// TwinCAT 3 PLC project PressTests
// Title: PressTests
// Company: fraktal-automation
// Author: fraktal-automation
// ProjectVersion: 0.1.0.1
// Description: Press example TcUnit gate - excluded from deployed runtime (Core 5.7).
// ProgramVersion: 3.1.4026.24
// libraries:
//   Tc2_Standard, * (Beckhoff Automation GmbH)
//   Tc2_System, * (Beckhoff Automation GmbH)
//   Tc2_Utilities, * (Beckhoff Automation GmbH)
//   Tc3_Module, * (Beckhoff Automation GmbH)
//   Fraktal_Core, 0.25.0.0 (fraktal-automation)
//   Tc2_MC2, * (Beckhoff Automation GmbH)
//   Fraktal_Modules, 0.11.0.3 (fraktal-automation)
//   TcUnit, * (www.tcunit.org)
// project tree:
//   PressTests/ PlcTask.TcTTO, PRG_PressTestRunner.TcPOU, FB_PressDemoUnit_Tests.TcPOU, FB_FaultRecovery_Tests.TcPOU
//   Fraktal_Press_Demo/01_PneumaticPress/DUTs/ ST_PneumaticPressParCfg.TcDUT, ST_PneumaticPressStationCfg.TcDUT, ST_PneumaticPressParCmd.TcDUT (not stored), ST_PneumaticPressOutCmd.TcDUT, ST_PneumaticPressOutImm.TcDUT, E_RenditionLanguage.TcDUT, ST_PressDemoReleaseConditions.TcDUT
//   Fraktal_Press_Demo/01_PneumaticPress/ PL_PressReasons.TcGVL, FB_PressDemoUnit.TcPOU
//   Fraktal_Press_Demo/01_PneumaticPress/Recipes/ FB_PressRecipeCatalog.TcPOU
//   Fraktal_Press_Demo/01_PneumaticPress/Release/ FB_PressDemoRelease.TcPOU, FB_LD_PressDemoRelease.TcPOU, FB_PressDemoReleaseState.TcPOU
//   Fraktal_Press_Demo/01_PneumaticPress/Sequences/ FB_PressDemoHome.TcPOU, FB_PressDemoAuto.TcPOU, FB_SFC_PressDemoAuto.TcPOU, FB_LD_PressDemoAuto.TcPOU, FB_PressDemoChangeover.TcPOU, FB_PressDemoLoadPosition.TcPOU
//   Fraktal_Press_Demo/01_PneumaticPress/Io/ GVL_PressFieldbus.TcGVL, FB_PressIoCatalog.TcPOU
// real-time tasks:
//   TASK PlcTask: cycle T#10ms, priority 20, ADS port 350

CONFIGURATION PressTests
    RESOURCE PLC ON TwinCAT3
        TASK PlcTask(INTERVAL := T#10ms, PRIORITY := 20);
        PROGRAM PRG_PressTestRunner WITH PlcTask : PRG_PressTestRunner;
    END_RESOURCE
END_CONFIGURATION

// ---- Fraktal_Press_Demo/01_PneumaticPress/DUTs/ST_PneumaticPressParCfg.TcDUT
// Core §3.8 ParCfg (SchemaVersion first; adding a member = schema change).
// v2 adds the §8.11 performance references: per-model ideal cycle (OEE
// Performance denominator, §8.5.1) and the WORK-time degradation baseline
// (§8.11.4(d); 0 = watch off).
//
// v3 REMOVES RequireTwoHandStart. It was recipe data in name only - every one of
// the four catalog records set it TRUE - and §3.8a's test is whether the value
// changes with the model. It does not: it answers whether this CELL's risk
// assessment demands a two-hand start, which is deployment data and now lives in
// ST_PneumaticPressStationCfg. A recipe that could switch it off would let a
// changeover quietly remove a required operator protection.
//
// TransferSettleTime deliberately STAYED. Its catalog values genuinely differ per
// model (80/100/120/150 ms): a heavier steel blank settles on the slide more
// slowly than a plastic one, so it is a fact about the part, not the mechanism.
TYPE ST_PneumaticPressParCfg :
STRUCT
    SchemaVersion       : UINT := 3;
    PressSettleTime     : TIME := T#500MS;
    TransferSettleTime  : TIME := T#100MS;
    IdealCycleMs        : UDINT := 0;    // §8.5.1 — 0 = Performance not computed
    BaselineWorkMs      : UDINT := 0;    // §8.11.4(d) — 0 = degradation watch off
END_STRUCT
END_TYPE

// ---- Fraktal_Press_Demo/01_PneumaticPress/DUTs/ST_PneumaticPressStationCfg.TcDUT
// Core §3.8a/§3.8b — what this PRESS is, as opposed to what the current product
// needs. Both members were assessed against one question: does the value change
// when the MODEL changes?
//
//   RequireTwoHandStart came OUT of ST_PneumaticPressParCfg. It was recipe data
//   in name only - all four catalog records set it TRUE - and it answers a
//   question about the CELL: does this installation's risk assessment demand a
//   two-hand start? A model recipe able to switch it off would let a changeover
//   quietly remove a required operator protection, which is not a decision a
//   product record should be able to take. (The certified two-hand evaluation
//   stays in TwinSAFE regardless, §9.8; this flag selects whether the AUTO cycle
//   WAITS for it, and can never weaken the safety function itself.)
//
//   StallGuardMs is the step guard for a step that declares no ExpectedTime
//   (§6.9). How long a pneumatic motion may take before it counts as stalled is
//   a fact about this machine's cylinders and air supply, not about the part.
//
// SchemaVersion is FIRST and mandatory (§3.8b). Version 0 means never written, so
// a first boot initializes silently; any other unrecognized version means a real
// image was rejected, and FB_ModuleBase.M_RestoreStationCfg reports it for the
// root to annunciate with this Unit's canonical path.
TYPE ST_PneumaticPressStationCfg :
STRUCT
    SchemaVersion       : UINT;    // 0 = never written; 1 = this layout
    RequireTwoHandStart : BOOL;    // cell risk-assessment policy, not recipe data
    StallGuardMs        : UDINT;   // §6.9 step guard when a step declares none
END_STRUCT
END_TYPE

// ---- Fraktal_Press_Demo/01_PneumaticPress/DUTs/ST_PneumaticPressOutCmd.TcDUT
TYPE ST_PneumaticPressOutCmd :
STRUCT
    // §3.12 — OutCmd is what a COMMAND PRODUCED, latched until the next command.
    // Both of these are genuine command results: a cycle ran, a changeover ran.
    // `Homed` used to live here and does not any more - being at the home position
    // is not something a command produced, it is something that is either true now
    // or not, so it is derived state (OutImm.Homed) recomputed every scan.
    CycleCompleted : BOOL;
    ChangeoverCompleted : BOOL;
END_STRUCT
END_TYPE

// ---- Fraktal_Press_Demo/01_PneumaticPress/DUTs/ST_PneumaticPressOutImm.TcDUT
TYPE ST_PneumaticPressOutImm :
STRUCT
    // Only facts the Unit DERIVES. A child's own state is read on the child
    // (PressRam.OutImm.Retracted, ...), never copied here under a second name (O9).
    //
    // §3.12 derived state: TRUE while the machine IS at its reference position.
    // As a latched command result it went on claiming "homed" after an operator
    // jogged an axis off home in MANUAL, because no sequence ran to clear it.
    Homed           : BOOL;
    // TRUE while a two-hand press would start a cycle: buttons armed, the control
    // domain ready, a part loaded and air present. Drives the pushbutton lamps.
    TwoHandStartReady : BOOL;
END_STRUCT
END_TYPE

// ---- Fraktal_Press_Demo/01_PneumaticPress/DUTs/E_RenditionLanguage.TcDUT
// Which language a parallel rendition of the same engineering is written in.
// The internal press bench carries the AUTO chain three times and the release
// engineering twice — the same behaviour in a second language is a
// demonstration of §5.5/§6.8 language parity, not §1.1 O9 duplication.
// FB_PressDemoUnit selects one of each; the compiler folds the branches the
// selection does not take, so the unselected renditions are inert.
//
// ONE type for both selections on purpose: a value has to mean the same
// language wherever it appears. The release engineering has no
// SEQUENTIAL_FUNCTION_CHART rendition — SFC is a sequence language and has
// nothing to say about a permissive — so that member is simply never selected
// there. The gap is deliberate; it is not an invitation to reuse the value for
// something else.
//
// The members are spelled out rather than abbreviated because 'ST' is a
// reserved word (the IL store operator). As an enumeration member it desyncs
// the parser and cascades misleading errors onto innocent lines (lint C2).
{attribute 'qualified_only'}
TYPE E_RenditionLanguage :
(
    STRUCTURED_TEXT           := 0,   // §6.8 reference form: CASE _step OF + M_Advance
    SEQUENTIAL_FUNCTION_CHART := 1,   // native XAE chart; sequences only
    LADDER_DIAGRAM            := 2    // rung-per-state integer machine over _step
) DINT;
END_TYPE

// ---- Fraktal_Press_Demo/01_PneumaticPress/DUTs/ST_PressDemoReleaseConditions.TcDUT
// Core §7.2/§3.12 - the press's named release conditions, as PUBLISHED.
// Filled every scan from whichever rendition RELEASE_LANGUAGE selects, so a
// browsing client always reads the conditions that are actually being
// evaluated. Before this, the ST component was the published one and was
// never evaluated while LADDER_DIAGRAM was selected: every flag sat at its
// initial FALSE whatever the machine was doing - state nobody computes,
// published as if it were a claim.
TYPE ST_PressDemoReleaseConditions :
STRUCT
    ModeStartAirPressureOk : BOOL;
    RamGuardClosed    : BOOL;
    RamSlideInside    : BOOL;
    RamDevicesHealthy : BOOL;
    RamAirPressureOk  : BOOL;
    RamTwoHandHeld    : BOOL;
    RamControlPowerOn : BOOL;
END_STRUCT
END_TYPE

// ---- Fraktal_Press_Demo/01_PneumaticPress/PL_PressReasons.TcGVL
{attribute 'qualified_only'}
// Core §8.8 band constants for THIS project: pneumatic press 12000-12999.
// Project codes deliberately sit outside the shipped registry, so a message
// raised with one keeps the severity and category the step chose.
VAR_GLOBAL CONSTANT
    PRESS_TWO_HAND_RELEASED : DINT := 12001;   // released mid-motion: cycle aborted, no damage
END_VAR

// ---- Fraktal_Press_Demo/01_PneumaticPress/Io/GVL_PressFieldbus.TcGVL
{attribute 'qualified_only'}
// Owner-local, bounded publication of the demo's physical CX2030 I/O tree.
// ST_IoChannel.Name is always the exact electrical-list/schematic tag.
VAR_GLOBAL
    {attribute 'OPC.UA.DA' := '1'}
    Topology : ST_FieldbusTopology;
END_VAR

// ---- PressTests/PRG_PressTestRunner.TcPOU
// Core 5.7 / TC3 5.7 - internal Press feature-bench integration gate.
// Split out of the aggregate Fraktal_Tests suite: TwinCAT rejects a Compile
// path containing '..', so a manifest inside Tests/ cannot reach the press
// sources in Examples/. These two suites therefore run from the example they
// exercise, against the SAME source objects that deploy (linked, never copied).
PROGRAM PRG_PressTestRunner
VAR
    PressDemoTests     : FB_PressDemoUnit_Tests;
    FaultRecoveryTests : FB_FaultRecovery_Tests;
END_VAR

TcUnit.RUN();

END_PROGRAM

// ---- PressTests/FB_PressDemoUnit_Tests.TcPOU
FUNCTION_BLOCK FB_PressDemoUnit_Tests EXTENDS TcUnit.FB_TestSuite
VAR
    Press : FB_PressDemoUnit;
    PressHal, DoorHal, SlideHal : ST_CylinderHal;
    TwoHandHal : ST_TwoHandHal;
    PowerHal : ST_PowerGroupHal;
    PartPresentHal : ST_DigitalInputHal;
    AirPressureHal : ST_AirPressureHal;
    PressSim, DoorSim, SlideSim : FB_CylinderSim;
    Recipe : FB_LocalRecipeProvider;
    Fast, Slow : ST_PneumaticPressParCfg;
    SlowModel : ST_ModelId;
    Domain : ST_ControlDomainStatus;
    Release : ST_ReleaseReport;
    Wired : BOOL;
    i : INT;
END_VAR

IF NOT Wired THEN
    Fast.PressSettleTime := T#0S; Fast.TransferSettleTime := T#0S;
    Fast.IdealCycleMs := 1000; Fast.BaselineWorkMs := 900;
    Slow.PressSettleTime := T#1200MS; Slow.TransferSettleTime := T#100MS;
    Slow.IdealCycleMs := 2500; Slow.BaselineWorkMs := 2200;
    Recipe.Register(ModelCode := '', RecipeKey := 'PneumaticPressUnit', pData := ADR(Fast), Size := SIZEOF(Fast));
    Recipe.Register(ModelCode := 'STEEL', RecipeKey := 'PneumaticPressUnit', pData := ADR(Slow), Size := SIZEOF(Slow));
    PressHal.RetractedFb := TRUE; DoorHal.RetractedFb := TRUE; SlideHal.RetractedFb := TRUE;
    Press.Setup(Name := 'Test.Press', PressHal := PressHal, DoorHal := DoorHal,
        SlideHal := SlideHal, TwoHandHal := TwoHandHal, PowerHal := PowerHal,
        PartPresentHal := PartPresentHal, AirPressureHal := AirPressureHal, Recipe := Recipe);
    PressSim.Setup(HalRef := PressHal, TravelTime := T#0S);
    DoorSim.Setup(HalRef := DoorHal, TravelTime := T#0S);
    SlideSim.Setup(HalRef := SlideHal, TravelTime := T#0S);
    PowerHal.SafetyPermit := TRUE; PowerHal.FieldbusHealthy := TRUE; PowerHal.PowerFeedback := TRUE;
    TwoHandHal.FieldbusHealthy := TRUE;
    PartPresentHal.Quality := TRUE; AirPressureHal.Quality := TRUE;
    Domain.Present := TRUE; Domain.Id := 'TEST-PRESS'; Domain.ReadyForStart := TRUE;
    Domain.Safety.Present := TRUE; Domain.Safety.AllSafe := TRUE;
    Domain.ControlPower.Present := TRUE; Domain.ControlPower.ControlOn := TRUE;
    Press.ControlDomain := Domain;
    PartPresentHal.Value := TRUE;
    AirPressureHal.LowPressure := FALSE; AirPressureHal.OperatingPressure := TRUE;
    Wired := TRUE;
END_IF
Model_changeover_is_transactional();
Start_release_enforces_operating_air();
Home_and_changeover_sequences_are_explicit();
Auto_cycle_returns_to_load_position();

METHOD Model_changeover_is_transactional
TEST('Model_changeover_is_transactional');
SlowModel.ModelCode := 'STEEL';
AssertTrue(Condition := Press.SetModel(Id := SlowModel), Message := 'stopped Unit accepts model changeover');
AssertTrue(Condition := Press.ParCfg.PressSettleTime = T#1200MS,
    Message := 'model-specific press dwell committed atomically');
AssertTrue(Condition := Press.Profiler.BaselineWorkMs = 2200,
    Message := 'model-specific profiler baseline committed through its owner API');
SlowModel.ModelCode := '';
AssertTrue(Condition := Press.SetModel(Id := SlowModel), Message := 'fallback recipe restores fast test model');
AssertTrue(Condition := Press.ParCfg.PressSettleTime = T#0S, Message := 'fallback recipe active');
AssertTrue(Condition := Press.Profiler.BaselineWorkMs = 900,
    Message := 'fallback profiler baseline follows the committed recipe');
TEST_FINISHED();
END_METHOD

// Press example of Core T10: an immediate mode-entry permissive is both
// explainable and enforced. Part/two-hand remain future AUTO step conditions.
METHOD Start_release_enforces_operating_air
TEST('Start_release_enforces_operating_air');
AssertTrue(Condition := Press.SetMode(Mode := E_Mode.AUTO), Message := 'AUTO selected for release test');
Press();
AirPressureHal.LowPressure := TRUE;
AirPressureHal.OperatingPressure := FALSE;
Press();
Press.ReleaseReportStart(Report := Release);
AssertFalse(Condition := Release.Released, Message := 'operating-air permissive is reported');
AssertFalse(Condition := Press.ReleaseConditions.ModeStartAirPressureOk,
    Message := 'project release component exposes the failed named condition');
AssertTrue(Condition := Release.Count >= 1, Message := 'release report names the failed condition');
AssertEquals_STRING(Expected := 'Test.Press', Actual := Release.Reasons[1].SourcePath,
    Message := 'release report retains press Unit ownership');
AssertFalse(Condition := Press.Start(), Message := 'reported operating-air permissive blocks Start');

AirPressureHal.LowPressure := FALSE;
AirPressureHal.OperatingPressure := TRUE;
Press();
Press.ReleaseReportStart(Report := Release);
AssertTrue(Condition := Release.Released, Message := 'release clears with operating air');
AssertTrue(Condition := Press.ReleaseConditions.ModeStartAirPressureOk,
    Message := 'project release component exposes the cleared named condition');
AssertTrue(Condition := Press.Start(), Message := 'Start accepts when the authoritative report releases');
Press.Stop();
Press();
TEST_FINISHED();
END_METHOD

METHOD Home_and_changeover_sequences_are_explicit
TEST('Home_and_changeover_sequences_are_explicit');
AssertTrue(Condition := Press.SetMode(Mode := E_Mode.HOME), Message := 'HOME is advertised');
Press();
AssertTrue(Condition := Press.Start(), Message := 'HOME starts through Unit lifecycle');
FOR i := 1 TO 20 DO
    PressSim(); DoorSim(); SlideSim(); Press();
END_FOR
AssertTrue(Condition := Press.OutImm.Homed, Message := 'HOME establishes load-safe position');
Press.Stop(); Press();
AssertTrue(Condition := Press.Start(),
    Message := 'HOME restarts without requiring an intervening mode change');
FOR i := 1 TO 20 DO
    PressSim(); DoorSim(); SlideSim(); Press();
END_FOR
AssertTrue(Condition := Press.OutImm.Homed,
    Message := 'repeated HOME receives a freshly reset finite chain');
Press.Stop(); Press();

AssertTrue(Condition := Press.SetMode(Mode := E_Mode.CHANGEOVER), Message := 'CHANGEOVER is advertised');
Press();
SlowModel.ModelCode := 'STEEL';
AssertTrue(Condition := Press.SetModel(Id := SlowModel), Message := 'selected recipe loads transactionally');
AirPressureHal.LowPressure := TRUE; AirPressureHal.OperatingPressure := FALSE;
Press();
Press.ReleaseReportStart(Report := Release);
AssertTrue(Condition := Release.Released, Message := 'CHANGEOVER entry does not require compressed air');
AssertTrue(Condition := Press.Start(), Message := 'guided CHANGEOVER starts without compressed air');
AirPressureHal.LowPressure := FALSE; AirPressureHal.OperatingPressure := TRUE;
PressSim(); DoorSim(); SlideSim(); Press();
AssertEquals_DINT(Expected := TO_DINT(E_HostEventKind.CHANGEOVER_STARTED),
    Actual := TO_DINT(Press.HostEvents.Ring[Press.HostEvents.RingHead].Kind),
    Message := 'host changeover starts on the accepted run edge');
FOR i := 1 TO 30 DO
    PressSim(); DoorSim(); SlideSim(); Press();
    IF Press.Decision.Prompt <> '' THEN Press.DecisionAnswer := 1; END_IF
END_FOR
AssertTrue(Condition := Press.OutCmd.ChangeoverCompleted,
    Message := 'CHANGEOVER completes only after operator confirmation');
AssertEquals_DINT(Expected := TO_DINT(E_HostEventKind.CHANGEOVER_DONE),
    Actual := TO_DINT(Press.HostEvents.Ring[Press.HostEvents.RingHead].Kind),
    Message := 'host changeover completes with the guided sequence');
AssertTrue(Condition := Press.Model.ModelCode = 'STEEL', Message := 'active model is published');
Press.Stop(); Press();
AssertTrue(Condition := Press.SetMode(Mode := E_Mode.AUTO), Message := 'AUTO remains available');
Press();
SlowModel.ModelCode := '';
AssertTrue(Condition := Press.SetModel(Id := SlowModel), Message := 'fast test recipe restored');
TEST_FINISHED();
END_METHOD

METHOD Auto_cycle_returns_to_load_position
VAR
    beforeRam, beforeDoor, beforeSlide : UDINT;
    firstGood : UDINT;
END_VAR
TEST('Auto_cycle_returns_to_load_position');
beforeRam := _M_CommandCount(pTiming := ADR(Press.PressRam.Timing), CommandId := 1);
beforeDoor := _M_CommandCount(pTiming := ADR(Press.Door.Timing), CommandId := 1);
beforeSlide := _M_CommandCount(pTiming := ADR(Press.PartSlide.Timing), CommandId := 1);
PartPresentHal.Value := FALSE;
AirPressureHal.LowPressure := TRUE; AirPressureHal.OperatingPressure := FALSE;
TwoHandHal.LeftPressed := FALSE; TwoHandHal.RightPressed := FALSE; TwoHandHal.SafeActive := FALSE;
Press();
TwoHandHal.LeftPressed := TRUE; TwoHandHal.RightPressed := TRUE; TwoHandHal.SafeActive := TRUE;
Press();
AssertTrue(Condition := Press.State = E_ExecState.READY,
    Message := 'two-hand edge is not cached without part and operating air');
TwoHandHal.LeftPressed := FALSE; TwoHandHal.RightPressed := FALSE; TwoHandHal.SafeActive := FALSE;
PartPresentHal.Value := TRUE;
AirPressureHal.LowPressure := FALSE; AirPressureHal.OperatingPressure := TRUE;
Press();
TwoHandHal.LeftPressed := TRUE; TwoHandHal.RightPressed := TRUE; TwoHandHal.SafeActive := TRUE;
FOR i := 1 TO 80 DO
    PressSim(); DoorSim(); SlideSim(); Press();
END_FOR
AssertTrue(Condition := Press.GoodCount > 0, Message := 'AUTO cycle records a good part');
AssertTrue(Condition := PressHal.RetractedFb, Message := 'ram returns up');
AssertTrue(Condition := DoorHal.RetractedFb, Message := 'door returns open');
AssertTrue(Condition := SlideHal.RetractedFb, Message := 'slide returns outside for unloading');
firstGood := Press.GoodCount;
TwoHandHal.LeftPressed := FALSE; TwoHandHal.RightPressed := FALSE; TwoHandHal.SafeActive := FALSE;
PressSim(); DoorSim(); SlideSim(); Press();
PressSim(); DoorSim(); SlideSim(); Press();
TwoHandHal.LeftPressed := TRUE; TwoHandHal.RightPressed := TRUE; TwoHandHal.SafeActive := TRUE;
FOR i := 1 TO 80 DO
    PressSim(); DoorSim(); SlideSim(); Press();
END_FOR
AssertEquals_UDINT(Expected := firstGood + 1, Actual := Press.GoodCount,
    Message := 'a fresh two-hand edge completes a second actual cycle');
AssertTrue(Condition := _M_CommandCount(pTiming := ADR(Press.PressRam.Timing), CommandId := 1) >= beforeRam + 2,
    Message := 'ram EXTEND completed anew in both cycles');
AssertTrue(Condition := _M_CommandCount(pTiming := ADR(Press.Door.Timing), CommandId := 1) >= beforeDoor + 2,
    Message := 'door EXTEND completed anew in both cycles');
AssertTrue(Condition := _M_CommandCount(pTiming := ADR(Press.PartSlide.Timing), CommandId := 1) >= beforeSlide + 2,
    Message := 'slide EXTEND completed anew in both cycles');
AssertTrue(Condition := PressHal.RetractedFb AND DoorHal.RetractedFb AND SlideHal.RetractedFb,
    Message := 'second cycle returns every cylinder to load position');
TEST_FINISHED();
END_METHOD

METHOD PRIVATE _M_CommandCount : UDINT
VAR_INPUT
    pTiming : POINTER TO ST_ModuleTiming;
    CommandId : DINT;
END_VAR
VAR
    rowIndex : INT;
END_VAR
_M_CommandCount := 0;
FOR rowIndex := 1 TO PL_Fraktal.MAX_CMD_STATS DO
    IF pTiming^.Rows[rowIndex].Id = CommandId THEN
        _M_CommandCount := pTiming^.Rows[rowIndex].Count;
        RETURN;
    END_IF
END_FOR
END_METHOD

END_FUNCTION_BLOCK

// ---- Fraktal_Press_Demo/01_PneumaticPress/FB_PressDemoUnit.TcPOU
// Project-owned Unit: pneumatic press + access door + transfer slide + two-hand request.
// Cylinder interlocks prevent the two documented collisions in AUTO and MANUAL.
// Certified E-stop, two-hand evaluation and safe valve outputs remain external.
FUNCTION_BLOCK FB_PressDemoUnit EXTENDS FB_UnitBase
VAR_INPUT
    ParCfg : ST_PneumaticPressParCfg;
    ParCmd : ST_PneumaticPressParCmd;
END_VAR
VAR_OUTPUT
    PressRam      : FB_CylinderCM;
    Door          : FB_CylinderCM;
    PartSlide     : FB_CylinderCM;
    TwoHand       : FB_TwoHandStartCM;
    PneumaticPower: FB_PowerGroupCM;
    PartPresentSensor : FB_DigitalInputCM;
    AirPressureMonitor : FB_AirPressureMonitorCM;
    // Jenny Science XENAX Xvi servo (Annex G, PLCopen Motion). NOT CABINET
    // HARDWARE - read the note on PartFeedAxis before looking for it there.
    PartFeed      : FB_AxisCM;
    // Project-owned, browseable condition state of the rendition that RUNS.
    ReleaseConditions : ST_PressDemoReleaseConditions;
    OutCmd        : ST_PneumaticPressOutCmd;
    OutImm        : ST_PneumaticPressOutImm;
END_VAR
VAR
    {attribute 'OPC.UA.DA' := '0'}
    _recipe : I_RecipeProvider;
    // The NC axis this Unit feeds parts with. Until an axis is actually linked
    // in the System Manager, _partFeedConfigured stays FALSE and the module is
    // never called: MC_Power against an unlinked AXIS_REF would otherwise run
    // every scan on a bench whose eight tests are green. Absent hardware is
    // absent, not silently pretended.
    //
    // WHAT THIS AXIS IS, AND IS NOT (2026-08-25). The delivered CX2030 cabinet
    // has NO SERVO. Its approved I/O list is five Beckhoff terminals
    // (=000+S-K010: EK1200 / EL1809 / EL2809 / EL6001 / EL9011 -- see
    // Specification/Reports/CX2030_PRESS_IO_MAPPING.md), and the part feeder in
    // that cabinet is PNEUMATIC: PartSlide above, driven by the digital outputs
    // _101K301A/_101K301B. Do not go looking for this axis on the cabinet bus.
    //
    // The drive behind it is a Jenny Science XENAX Xvi (vendor #x557, product
    // #x7508) on a SECOND EtherCAT device, =000+S-A620 (EtherCAT), kept in its
    // own XTI beside the cabinet's. It is outside the press entirely and stands
    // in for a feed axis so a real process can be simulated against real motion
    // hardware. Anything it teaches (S3.8c) or persists (S3.8b) is BENCH data,
    // not commissioning data for the press -- which is why =000+S-A610-A1
    // (EtherCAT).xti, the faithful record of the delivered cabinet, does not
    // mention it and must not be made to.
    {attribute 'OPC.UA.DA' := '0'}
    PartFeedAxis : AXIS_REF;
    _partFeedConfigured : BOOL;
    _partFeedArmed : BOOL;             // last arming attempt's result (S5.6: no discarded return)
    // §10.5.1 - the project I/O catalog owns the approved channel identity join
    // (§10.2.1), so it, not this Unit, resolves a force request to a physical
    // channel. Absent = no force routing, which is the fail-closed default.
    {attribute 'OPC.UA.DA' := '0'}
    _ioCatalog : REFERENCE TO FB_PressIoCatalog;
    _parCfgStaged : ST_PneumaticPressParCfg;
    // §3.8a - the ParCfg last applied (commit or accepted edit); a difference is an
    // edit of the active model's recipe to take effect and to write back.
    {attribute 'OPC.UA.DA' := '0'}
    _parCfgApplied : ST_PneumaticPressParCfg;
    _recipePrepared : BOOL;
    _startLatched : BOOL;
    _powerRequestPending : BOOL;
    _powerTargetOn : BOOL;
    {attribute 'OPC.UA.DA' := '0'}
    _homeSequence : FB_PressDemoHome;       // §6.8 ST chain on FB_SequenceBase owns HOME steps
    {attribute 'OPC.UA.DA' := '0'}
    _changeoverSequence : FB_PressDemoChangeover;
    // §6.8 / O2 — the SAME AUTO chain in all three permitted languages. This is a
    // demo bench: carrying three renditions is the point (O2 says sequences and
    // interlocks may be ST, SFC or Ladder), not something a real project would do.
    // AUTO_SEQUENCE_LANGUAGE below picks which one the Unit binds and runs; the
    // other two are inert. They are excluded from OPC UA for the same reason the
    // bound one is: a chain is not a module and publishes no Status.
    {attribute 'OPC.UA.DA' := '0'}
    _autoSequence : FB_PressDemoAuto;
    {attribute 'OPC.UA.DA' := '0'}
    _sfcAutoSequence : FB_SFC_PressDemoAuto;
    {attribute 'OPC.UA.DA' := '0'}
    _ldAutoSequence : FB_LD_PressDemoAuto;
    // §7.2 / O2 — the SAME release engineering in a second language. Only the
    // rendition RELEASE_LANGUAGE selects is set up, evaluated, and allowed to
    // write the directional permits and the release report; the other is inert.
    // Neither rendition is published itself: the selected one fills
    // ReleaseConditions (a VAR_OUTPUT above) every scan, so the browseable
    // record is always the one being evaluated. Publishing the ST instance
    // directly left it frozen at FALSE whenever LD was selected (§3.12).
    {attribute 'OPC.UA.DA' := '0'}
    _stReleaseConditions : FB_PressDemoRelease;
    {attribute 'OPC.UA.DA' := '0'}
    _ldReleaseConditions : FB_LD_PressDemoRelease;
END_VAR
VAR PERSISTENT
    // §3.8b - this station's deployment data. PERSISTENT is the BACKING, not the
    // architecture: the values are reached as (Scope, WriteKey) capabilities like
    // every other editable value, never as an aggregate copied in and out.
    _station : ST_PneumaticPressStationCfg;
END_VAR
VAR CONSTANT
    // §3.8b - layout version of the retained image above. Bump it when a member
    // is added, and the old image is rejected and annunciated instead of read by
    // field position.
    PRESS_STATIONCFG_SCHEMA : UINT := 1;
    // §3.8 - the longest settle times a recipe may hold. ONE source for the check
    // a changeover applies (PrepareRecipe) and the range an edit is offered
    // (the PAR_CFG registration), so an edit can never store what a changeover
    // would refuse.
    RECIPE_MAX_PRESS_SETTLE_MS    : UDINT := 30000;
    RECIPE_MAX_TRANSFER_SETTLE_MS : UDINT := 5000;
    // The provider key of this Unit's recipe record: loaded at a changeover and
    // edited per model through the same key (§3.8a).
    PRESS_RECIPE_KEY : STRING(80) := 'PneumaticPressUnit';
    // Which rendition of the AUTO chain runs. VAR CONSTANT on purpose, like the
    // §6.0 commissioning gates in MAIN: switching language is a source edit plus a
    // download, never an online write. The compiler folds the unselected branches.
    //   STRUCTURED_TEXT           -> FB_PressDemoAuto
    //   SEQUENTIAL_FUNCTION_CHART -> FB_SFC_PressDemoAuto
    //   LADDER_DIAGRAM            -> FB_LD_PressDemoAuto
    AUTO_SEQUENCE_LANGUAGE : E_RenditionLanguage := E_RenditionLanguage.LADDER_DIAGRAM;
    // Which rendition of the release/interlock logic is evaluated, on the same
    // terms and from the same type, so a value means the same language in both
    // selections. There is no SEQUENTIAL_FUNCTION_CHART rendition here: SFC is a
    // sequence language and has nothing to say about a permissive, so that
    // member is simply never selected rather than being given a second meaning.
    //   STRUCTURED_TEXT -> FB_PressDemoRelease
    //   LADDER_DIAGRAM  -> FB_LD_PressDemoRelease
    RELEASE_LANGUAGE : E_RenditionLanguage := E_RenditionLanguage.LADDER_DIAGRAM;
END_VAR

Cyclic();

// §7.8 mode-entry release owned by this Unit. The base Start method consumes the
// same report the HMI displays, so this condition cannot become explanation-only.
METHOD PROTECTED _M_AppendInterlocks
VAR_IN_OUT
    Report : ST_ReleaseReport;
END_VAR
IF ModeActive <> E_Mode.CHANGEOVER THEN
IF RELEASE_LANGUAGE = E_RenditionLanguage.LADDER_DIAGRAM THEN
    _ldReleaseConditions.M_AppendStart(Report := Report);
ELSE
    _stReleaseConditions.M_AppendStart(Report := Report);
END_IF
END_IF
END_METHOD

METHOD PROTECTED _M_AppendManualInterlocks
VAR_INPUT
    TargetPath : STRING(255);
    Value : DINT;
END_VAR
VAR_IN_OUT
    Report : ST_ReleaseReport;
END_VAR
IF RELEASE_LANGUAGE = E_RenditionLanguage.LADDER_DIAGRAM THEN
    _ldReleaseConditions.M_AppendManual(TargetPath := TargetPath, Value := Value,
        PressRam := PressRam, Door := Door, PartSlide := PartSlide, Report := Report);
ELSE
    _stReleaseConditions.M_AppendManual(TargetPath := TargetPath, Value := Value,
        PressRam := PressRam, Door := Door, PartSlide := PartSlide, Report := Report);
END_IF
END_METHOD

// Clear state that must not survive init, mode entry, or either abort path. The
// base already restarts the chains and clears their decision (§6.8); this is the
// Unit's OWN state. OnCommandStart deliberately does not call this: a physical
// start pulse may have been latched one scan before the Execute edge is consumed.
METHOD PROTECTED _M_ClearModeTransitionState
_startLatched := FALSE;
END_METHOD

// Thin mode router. Each supported sequence is a named method in the Unit tree.
METHOD PROTECTED _M_Dispatch
CASE ModeActive OF
    E_Mode.AUTO:
        _M_SequenceAuto();
    E_Mode.HOME:
        _M_SequenceHome();
    E_Mode.CHANGEOVER:
        _M_SequenceChangeover();
    E_Mode.MANUAL:
        _M_Fault(E_Reason.UNSUPPORTED_COMMAND, 'project.error.pressManualHasNoSequence');
ELSE
    _M_Fault(E_Reason.UNSUPPORTED_COMMAND, 'project.error.pressModeHasNoSequence');
END_CASE
END_METHOD

// §10.2.1 — inject this station's I/O catalog so §10.5.1 force requests can be
// resolved against the approved engineering-data join instead of against a
// second copy of the channel map. Wired once by the composition root.
METHOD SetIoCatalog
VAR_INPUT
    Catalog : REFERENCE TO FB_PressIoCatalog;
END_VAR
_ioCatalog REF= Catalog;
END_METHOD

// §10.5.1 — resolve an accepted force request onto a physical output channel.
// FB_UnitBase.ForceChannel has already proved the §7.7 MANUAL access level, the
// §7.5 OUTPUT_FORCING build gate, and that this Unit is idle in MANUAL; the
// catalog then proves what only it knows — that the path names a channel of THIS
// root, that it is an OUTPUT, and that the project marked it forceable.
METHOD PROTECTED _M_RouteForceChannel : BOOL
VAR_INPUT
    ChannelPath : STRING(255);
    Force       : BOOL;
    BoolText    : STRING(255);
    AnalogText  : STRING(160);
END_VAR
_M_RouteForceChannel := FALSE;
IF NOT __ISVALIDREF(_ioCatalog) THEN
    RETURN;
END_IF
// The transported value is text (the mailbox carries no variant), so a malformed
// payload must decode to a defined value rather than to whatever the converter
// leaves behind: anything that is not exactly 'true' is FALSE (§5.6).
_M_RouteForceChannel := _ioCatalog.M_RouteForce(ChannelPath := ChannelPath,
    OwnerRootPath := _name, Force := Force,
    BoolValue := (BoolText = 'true'),
    AnalogValue := STRING_TO_REAL(AnalogText));
END_METHOD

// Wiring-only AUTO adapter. Every production command, wait, timer, decision,
// traceability action, and transition lives in the §6.8 chain.
METHOD PROTECTED _M_SequenceAuto
// An ST chain's body is a method (M_Run); an SFC or LD chain's body IS the chart,
// so the instance itself is the call. That asymmetry is the language difference,
// not an inconsistency to normalise away.
IF AUTO_SEQUENCE_LANGUAGE = E_RenditionLanguage.LADDER_DIAGRAM THEN
    _ldAutoSequence();
ELSIF AUTO_SEQUENCE_LANGUAGE = E_RenditionLanguage.SEQUENTIAL_FUNCTION_CHART THEN
    _sfcAutoSequence();
ELSE
    _autoSequence.M_Run();
END_IF
END_METHOD

// Wiring-only CHANGEOVER adapter. The §6.8 chain owns model validation, safe
// positioning, the operator decision, and completion logic.
METHOD PROTECTED _M_SequenceChangeover
_changeoverSequence.M_Run();
END_METHOD

// Wiring-only HOME adapter. OnCommandStart owns the reset edge; the sequence POU
// owns every process step and terminal action.
METHOD PROTECTED _M_SequenceHome
_homeSequence.M_Run();
END_METHOD

METHOD PROTECTED _M_Supports : BOOL
VAR_INPUT
    Mode : E_Mode;
END_VAR
_M_Supports := (Mode = E_Mode.AUTO) OR (Mode = E_Mode.MANUAL)
    OR (Mode = E_Mode.HOME) OR (Mode = E_Mode.CHANGEOVER);
END_METHOD

// §3.4.2 — the press paces every motion boundary through _M_StepGate, so
// SINGLE_STEP and HOLD_TO_RUN are supported (NON-SAFETY pacing; interlocks
// and the certified safety layer are unaffected).
METHOD PROTECTED _M_SupportsRunStyle : BOOL
VAR_INPUT
    Style : E_RunStyle;
END_VAR
_M_SupportsRunStyle := (Style = E_RunStyle.CONTINUOUS)
    OR (Style = E_RunStyle.SINGLE_STEP) OR (Style = E_RunStyle.HOLD_TO_RUN);
END_METHOD

// One safe-stop wiring point shared by normal and error-state abort transitions.
METHOD PROTECTED _M_WithdrawSequenceOutputs
PressRam.WithdrawOutputs();
Door.WithdrawOutputs();
PartSlide.WithdrawOutputs();
PressRam.Execute := FALSE;
Door.Execute := FALSE;
PartSlide.Execute := FALSE;
END_METHOD

METHOD AbortRecipe
SUPER^.AbortRecipe();
_recipePrepared := FALSE;
END_METHOD

METHOD CommitRecipe
SUPER^.CommitRecipe();
IF _recipePrepared THEN
    ParCfg := _parCfgStaged;
    // §8.11 performance references follow the model: OEE Performance denominator
    // and the WORK-time degradation baseline are per-recipe engineering data.
    Oee.IdealCycleMs := ParCfg.IdealCycleMs;
    Profiler.M_SetBaselineWork(WorkMs := ParCfg.BaselineWorkMs);
    _parCfgApplied := ParCfg;
END_IF
_recipePrepared := FALSE;
END_METHOD

// §3.10.2 — base walk (Unit facets + all child modules), then the project-owned
// fieldbus topology identity, from the I/O catalog that owns it (SetIoCatalog):
// its static members are OPC.UA.DA=0 and reach the HMI only through this manifest.
METHOD M_AppendConfig : BOOL
VAR_INPUT
    Pager : REFERENCE TO FB_ConfigPager;
END_VAR
M_AppendConfig := SUPER^.M_AppendConfig(Pager := Pager);
IF __ISVALIDREF(_ioCatalog) THEN
    _ioCatalog.M_AppendTopologyConfig(Pager := Pager);
END_IF
END_METHOD

METHOD PROTECTED OnAbort : DINT
OnAbort := SUPER^.OnAbort();
_M_PartAborted();                    // §3.16.3: the part leaves without a valid result
_M_WithdrawSequenceOutputs();
_M_ClearModeTransitionState();
_powerTargetOn := FALSE;
_powerRequestPending := TRUE;
END_METHOD

// Error-state Abort is a deliberate recovery action but does not clear ERROR.
METHOD PROTECTED OnAbortInError : DINT
OnAbortInError := SUPER^.OnAbortInError();
_M_WithdrawSequenceOutputs();
_M_ClearModeTransitionState();
_powerTargetOn := FALSE;
_powerRequestPending := TRUE;
END_METHOD

// The press's restart policy (§6.9(d)): every accepted Start gets a fresh mode
// chain, including a repeated HOME/CHANGEOVER run that does not pass through
// another mode change. Resuming where an error stopped is the other legitimate
// choice; this station does not make it.
METHOD PROTECTED OnCommandStart : DINT
OnCommandStart := SUPER^.OnCommandStart();
_M_RestartSequences();
END_METHOD

METHOD PROTECTED OnCyclic : DINT
VAR
    started : BOOL;
END_VAR
OnCyclic := SUPER^.OnCyclic();
// §3.8b/§3.12 — the step guard is DERIVED from the station value every scan, not
// latched at Setup. An operator who edits press.stallGuardMs gets the new guard
// on the next step, and the published StallTime can never disagree with the
// configuration it came from.
StallTime := UDINT_TO_TIME(_station.StallGuardMs);
// §3.8a - an accepted edit of the ACTIVE model's recipe lands in ParCfg (the base
// has already saved it to the model's record). The performance references follow
// it, as they do at a changeover.
IF MEMCMP(ADR(ParCfg), ADR(_parCfgApplied), SIZEOF(ParCfg)) <> 0 THEN
    Oee.IdealCycleMs := ParCfg.IdealCycleMs;
    Profiler.M_SetBaselineWork(WorkMs := ParCfg.BaselineWorkMs);
    _parCfgApplied := ParCfg;
END_IF
// §7.2.1/§6.1 - a cylinder cannot move without air, so air is each cylinder's own
// process condition. Lost mid-stroke, the cylinder HOLDS - outputs off, resumes by
// itself when pressure returns - and the Unit rolls the hold up by name. Nothing
// to reset: the process restores this condition, it is not a defect.
PressRam.SetAreaSafe(Ok := AirPressureMonitor.OutImm.PressureOk,
    DescriptionKey := 'project.interlock.pressRequiresAirPressure');
Door.SetAreaSafe(Ok := AirPressureMonitor.OutImm.PressureOk,
    DescriptionKey := 'project.interlock.pressRequiresAirPressure');
PartSlide.SetAreaSafe(Ok := AirPressureMonitor.OutImm.PressureOk,
    DescriptionKey := 'project.interlock.pressRequiresAirPressure');
// Project release engineering is a separate visible component. It owns the
// functional collision permits and mode-entry conditions consumed below.
IF RELEASE_LANGUAGE = E_RenditionLanguage.LADDER_DIAGRAM THEN
    _ldReleaseConditions.M_Evaluate(PressRam := PressRam, Door := Door, PartSlide := PartSlide,
        TwoHand := TwoHand, PneumaticPower := PneumaticPower,
        AirPressure := AirPressureMonitor);
    _ldReleaseConditions.M_PublishTo(Conditions := ReleaseConditions);
ELSE
    _stReleaseConditions.M_Evaluate(PressRam := PressRam, Door := Door, PartSlide := PartSlide,
        TwoHand := TwoHand, PneumaticPower := PneumaticPower,
        AirPressure := AirPressureMonitor);
    _stReleaseConditions.M_PublishTo(Conditions := ReleaseConditions);
END_IF

// S1.1 O1 - the axis ARMS ITSELF on the first scan a real NC axis is behind
// it, rather than through a call a composition root has to remember. Forgetting
// such a call produces a silently dead module, which is exactly the class of
// defect the objective says to drive from a path the application already takes.
// ConfigurePartFeedAxis is idempotent and fails closed, so calling it until it
// succeeds costs one comparison per scan on a bench with no drive.
IF NOT _partFeedConfigured THEN
    // THIS^ is required: an unqualified same-FB call resolves only when its
    // return value is discarded, and this one is not (C0009/C0035 otherwise).
    _partFeedArmed := THIS^.ConfigurePartFeedAxis(AxisRef := PartFeedAxis);
END_IF
// The feed axis runs only once an NC axis has been linked (S10.6). Its
// conditions are re-driven every scan so a manual move obeys the same rule as
// a sequenced one (S7.2).
//
// The module itself is NOT called here: ConfigurePartFeedAxis registers it as a
// child, and _M_TickChildren already ticks every registered child from
// SUPER^.OnCyclic above. Calling it here as well would run the whole S6.1
// lifecycle twice per scan.
// No conditions are driven here any more. Both that used to be - the press's
// pneumatic power and its ram guard - describe the PRESS, and the Xvi is
// physically outside it on a separate EtherCAT device. Gating a bench servo on
// whether a pneumatic valve zone somewhere else is energised is not an
// interlock, it is an unrelated fact that happens to block motion, and S7.2.1
// says a condition is defined at the module with enough semantic context to own
// it. This Unit has none for that drive.

// Latch access-gated Unit requests, then observe one full Execute-low scan before
// starting another power-group command (PLCopen edge discipline).
IF ControlOffRequest THEN
    _powerTargetOn := FALSE;
    _powerRequestPending := TRUE;
ELSIF ControlOnRequest THEN
    _powerTargetOn := TRUE;
    _powerRequestPending := TRUE;
END_IF
IF PneumaticPower.Done OR PneumaticPower.Error OR PneumaticPower.Aborted THEN
    PneumaticPower.Execute := FALSE;
ELSIF _powerRequestPending AND NOT PneumaticPower.Execute
AND (PneumaticPower.State = E_ExecState.READY) THEN
    PneumaticPower.Abort := FALSE;
    IF _powerTargetOn THEN
        PneumaticPower.Command := E_PowerGroupCommand.POWER_ON;
    ELSE
        PneumaticPower.Command := E_PowerGroupCommand.POWER_OFF;
    END_IF
    PneumaticPower.Execute := TRUE;
    _powerRequestPending := FALSE;
END_IF

// A physical two-hand edge starts AUTO from READY, or releases a running Unit's
// two-hand wait. Start() is asked unconditionally: its release report is the whole
// start predicate and names whatever refuses it (§7.2.1, §7.8). What IS qualified
// is the start LATCH: a press counts only when the part and the air that the N100
// wait also names are already there, so a press made before the part was loaded
// can never start the stroke when the part arrives. N100 shows what it waits for.
IF TwoHand.OutImm.StartPulse THEN
    IF ModeActive = E_Mode.AUTO THEN
        IF State = E_ExecState.BUSY THEN
            started := TRUE;
        ELSE
            started := Start();
        END_IF
        _startLatched := started
            AND PartPresentSensor.OutImm.Value AND PartPresentSensor.OutImm.Quality
            AND AirPressureMonitor.OutImm.PressureOk;
    ELSE
        _startLatched := FALSE;
    END_IF
END_IF
IF PneumaticPower.Error AND (State = E_ExecState.BUSY) THEN
    _M_RollupFault();
END_IF
// §3.12 — ONE derivation, published under the name the operator knows and read
// by everything that needs the fact (§1.1 O9: derived, never duplicated). It is a
// state, not a command result: it stops being true the moment a cylinder leaves
// the position, including in MANUAL where no sequence runs to clear anything.
// _M_State publishes it on the generic flag table with the moment it last changed,
// so the HMI can render it without knowing this module type.
OutImm.Homed := _M_State(Idx := 1, Key := 'project.state.pressAtLoadPosition',
    Ok := Door.OutImm.Retracted AND NOT Door.OutImm.Extended
      AND PartSlide.OutImm.Retracted AND NOT PartSlide.OutImm.Extended
      AND PressRam.OutImm.Retracted AND NOT PressRam.OutImm.Extended);
// The pushbutton lamps' condition, derived here - where the facts live - so the
// composition root only maps it to the output (§10.2.1).
OutImm.TwoHandStartReady := _M_State(Idx := 2, Key := 'project.state.pressTwoHandStartReady',
    Ok := TwoHand.OutImm.Armed AND ControlDomain.ReadyForStart
      AND PartPresentSensor.OutImm.Value AND PartPresentSensor.OutImm.Quality
      AND AirPressureMonitor.OutImm.PressureOk);
END_METHOD

// First operational scan: initialize application-owned mode-chain state.
METHOD PROTECTED OnInit : DINT
OnInit := SUPER^.OnInit();
_M_ClearModeTransitionState();
END_METHOD

// Mode-entry wiring only. Step behavior remains in the selected sequence POU.
METHOD PROTECTED OnModeChanged : DINT
VAR_INPUT
    NewMode : E_Mode;
    OldMode : E_Mode;
END_VAR
OnModeChanged := SUPER^.OnModeChanged(
    NewMode := NewMode, OldMode := OldMode);
_M_ClearModeTransitionState();
END_METHOD

// An operator reset is recovering this Unit: put the application back to the same
// safe wiring an error-state abort establishes, so the reset the operator presses at
// the panel needs no separate Stop/Abort first. The base then releases the run
// command and the children's commands, so the next HOME gets a genuine command edge.
// Unlike the abort paths this does NOT touch control power in either direction: it
// never requests Control On (§9.8 forbids self-resume), and it must not request
// Control Off either — powering down a healthy control circuit would make the
// operator re-enable it before HOME could run, i.e. reintroduce the multi-action
// recovery this reset exists to remove. Power stays where the operator put it.
METHOD PROTECTED OnOperatorReset : DINT
OnOperatorReset := SUPER^.OnOperatorReset();
_M_WithdrawSequenceOutputs();
_M_RestartSequences();                // this station restarts after a reset (§6.9(d))
_M_ClearModeTransitionState();
END_METHOD

METHOD PrepareRecipe : BOOL
VAR_INPUT
    Model : ST_ModelId;
END_VAR
IF _recipe = 0 THEN
    _parCfgStaged := ParCfg;
    _recipePrepared := TRUE;
ELSIF _recipe.Load(ModelCode := Model.ModelCode, RecipeKey := PRESS_RECIPE_KEY, pParCfg := ADR(_parCfgStaged), Size := SIZEOF(_parCfgStaged)) THEN
    IF (TIME_TO_UDINT(_parCfgStaged.PressSettleTime) > RECIPE_MAX_PRESS_SETTLE_MS)
    OR (TIME_TO_UDINT(_parCfgStaged.TransferSettleTime) > RECIPE_MAX_TRANSFER_SETTLE_MS) THEN
        _M_Fault(E_Reason.RECIPE_INVALID, 'project.error.pressRecipeInvalid');
        _recipePrepared := FALSE;
        PrepareRecipe := FALSE;
        RETURN;
    END_IF
    _recipePrepared := TRUE;
ELSE
    _M_Fault(E_Reason.RECIPE_INVALID, 'std.error.recipeSchemaInvalid');
    _recipePrepared := FALSE;
    PrepareRecipe := FALSE;
    RETURN;
END_IF
PrepareRecipe := SUPER^.PrepareRecipe(Model := Model);
IF NOT PrepareRecipe THEN _recipePrepared := FALSE; END_IF
END_METHOD

// Application-only seam for ordinary hardwired Control On/Off buttons.
// It is a method (not OPC UA data), so HMI writes still use the access-gated
// ReqControlOn/ReqControlOff contract. The power CM rechecks safety and health.
METHOD RequestLocalControl : BOOL
VAR_INPUT
    ControlOn : BOOL;
END_VAR
_powerTargetOn := ControlOn;
_powerRequestPending := TRUE;
RequestLocalControl := TRUE;
END_METHOD

METHOD Setup : BOOL
VAR_INPUT
    Name : STRING(80);
    PressHal : REFERENCE TO ST_CylinderHal;
    DoorHal : REFERENCE TO ST_CylinderHal;
    SlideHal : REFERENCE TO ST_CylinderHal;
    TwoHandHal : REFERENCE TO ST_TwoHandHal;
    PowerHal : REFERENCE TO ST_PowerGroupHal;
    PartPresentHal : REFERENCE TO ST_DigitalInputHal;
    AirPressureHal : REFERENCE TO ST_AirPressureHal;
    Recipe : I_RecipeProvider;
END_VAR
VAR
    InitialModel : ST_ModelId;
    Ok : BOOL;
END_VAR
_M_SetName(Name);
_M_SetPresentation(DisplayNameKey := 'project.module.pneumaticPress.name', DescriptionKey := 'project.module.pneumaticPress.description', TypeKey := 'project.moduleType.pneumaticPress');
_recipe := Recipe;
Ok := PressRam.Setup(Name := CONCAT(Name, '.PressRam'), HalRef := PressHal, Recipe := 0);
Ok := Door.Setup(Name := CONCAT(Name, '.Door'), HalRef := DoorHal, Recipe := 0) AND Ok;
Ok := PartSlide.Setup(Name := CONCAT(Name, '.PartSlide'), HalRef := SlideHal, Recipe := 0) AND Ok;
Ok := TwoHand.Setup(Name := CONCAT(Name, '.TwoHand'), HalRef := TwoHandHal) AND Ok;
Ok := PneumaticPower.Setup(Name := CONCAT(Name, '.PneumaticPower'), HalRef := PowerHal) AND Ok;
Ok := PartPresentSensor.Setup(Name := CONCAT(Name, '.PartPresentSensor'),
    HalRef := PartPresentHal, DisplayNameKey := 'project.module.partPresentSensor.name',
    DescriptionKey := 'project.module.partPresentSensor.description') AND Ok;
Ok := AirPressureMonitor.Setup(Name := CONCAT(Name, '.AirPressureMonitor'),
    HalRef := AirPressureHal) AND Ok;
IF RELEASE_LANGUAGE = E_RenditionLanguage.LADDER_DIAGRAM THEN
    Ok := _ldReleaseConditions.Setup(UnitPath := Name) AND Ok;
ELSE
    Ok := _stReleaseConditions.Setup(UnitPath := Name) AND Ok;
END_IF
Ok := _homeSequence.Setup(Host := THIS^, PressRam := PressRam, Door := Door,
    PartSlide := PartSlide, OutCmd := OutCmd) AND Ok;
Ok := _changeoverSequence.Setup(Host := THIS^, PressRam := PressRam, Door := Door,
    PartSlide := PartSlide, OutCmd := OutCmd, Model := Model) AND Ok;
// Only the selected rendition is attached: M_Attach registers the chain with the
// Unit, so attaching all three would put three chains on one step pointer.
// §3.8b restore, BEFORE the chains are set up: they take _station by reference
// and the first scan must already see either the commissioned values or the
// declared defaults, never a half-initialized image. The rule itself lives in
// FB_ModuleBase - this type supplies only what is genuinely its own, which is
// what its defaults are.
IF NOT M_RestoreStationCfg(pVersion := ADR(_station.SchemaVersion),
        SchemaVersion := PRESS_STATIONCFG_SCHEMA) THEN
    // Fail-safe defaults: two-hand REQUIRED (a lost risk-assessment policy must
    // never come back as the permissive one), and the framework's own 30 s
    // stall guard.
    _station.RequireTwoHandStart := TRUE;
    _station.StallGuardMs := 30000;
END_IF
IF AUTO_SEQUENCE_LANGUAGE = E_RenditionLanguage.LADDER_DIAGRAM THEN
    Ok := _ldAutoSequence.Setup(Host := THIS^, PressRam := PressRam, Door := Door,
        PartSlide := PartSlide, TwoHand := TwoHand, PartPresentSensor := PartPresentSensor,
        AirPressureMonitor := AirPressureMonitor, ParCfg := ParCfg,
        StationCfg := _station, OutCmd := OutCmd,
        StartLatched := _startLatched) AND Ok;
ELSIF AUTO_SEQUENCE_LANGUAGE = E_RenditionLanguage.SEQUENTIAL_FUNCTION_CHART THEN
    Ok := _sfcAutoSequence.Setup(Host := THIS^, PressRam := PressRam, Door := Door,
        PartSlide := PartSlide, TwoHand := TwoHand, PartPresentSensor := PartPresentSensor,
        AirPressureMonitor := AirPressureMonitor, ParCfg := ParCfg,
        StationCfg := _station, OutCmd := OutCmd,
        StartLatched := _startLatched) AND Ok;
ELSE
    Ok := _autoSequence.Setup(Host := THIS^, PressRam := PressRam, Door := Door,
        PartSlide := PartSlide, TwoHand := TwoHand, PartPresentSensor := PartPresentSensor,
        AirPressureMonitor := AirPressureMonitor, ParCfg := ParCfg,
        StationCfg := _station, OutCmd := OutCmd,
        StartLatched := _startLatched) AND Ok;
END_IF
PneumaticPower.ParCfg.Kind := E_PowerGroupKind.VALVE_ZONE;
PneumaticPower.ParCfg.RequiredForControl := TRUE;
PneumaticPower.ParCfg.FieldbusLossReaction := E_FieldbusLossReaction.CONTROL_OFF;
Ok := _M_Register(PressRam) AND Ok;
Ok := _M_Register(Door) AND Ok;
Ok := _M_Register(PartSlide) AND Ok;
Ok := _M_Register(TwoHand) AND Ok;
Ok := _M_Register(PneumaticPower) AND Ok;
Ok := _M_Register(PartPresentSensor) AND Ok;
Ok := _M_Register(AirPressureMonitor) AND Ok;
// §3.8a/§3.10.2 - the two deployment values become editable CAPABILITIES. That
// registration, not publication and not DATA_WRITE, is what makes them writable,
// and it is also what puts them into a station parameter set: SaveConfigSet walks
// the same registry (§3.8b), so a value registered here needs no separate line
// anywhere to be saved, listed, exported and restored.
Ok := M_RegisterConfigFlag(Key := 'press.requireTwoHandStart',
    Item := 'StationCfg/RequireTwoHandStart',
    LabelKey := 'project.config.pressRequireTwoHandStart',
    Kind := E_ConfigKind.STATION_CFG, pTarget := ADR(_station.RequireTwoHandStart),
    RequiresReady := TRUE) AND Ok;
Ok := M_RegisterConfigNumber(Key := 'press.stallGuardMs',
    Item := 'StationCfg/StallGuardMs',
    LabelKey := 'project.config.pressStallGuardMs', Unit := E_EngUnit.MILLISECOND,
    Kind := E_ConfigKind.STATION_CFG, Storage := E_ConfigStorage.AS_UDINT,
    pTarget := ADR(_station.StallGuardMs), Minimum := 1000.0, Maximum := 600000.0,
    RequiresReady := TRUE) AND Ok;
// §3.8a - model data, PAR_CFG, over this Unit's recipe record. Registering the
// record makes these values editable for EVERY model in the catalog, and the base
// writes each edit back to that model's record. The ranges are the RECIPE_MAX_*
// constants PrepareRecipe also enforces.
IF Recipe <> 0 THEN
    Ok := M_RegisterModelData(pData := ADR(ParCfg), Size := SIZEOF(ParCfg),
        RecipeKey := PRESS_RECIPE_KEY, Provider := Recipe) AND Ok;
END_IF
Ok := M_RegisterConfigDuration(Key := 'press.recipe.pressSettle',
    Item := 'ParCfg/PressSettleTime', LabelKey := 'project.config.pressSettleTime',
    Kind := E_ConfigKind.PAR_CFG, pTarget := ADR(ParCfg.PressSettleTime),
    MinimumMs := 0, MaximumMs := RECIPE_MAX_PRESS_SETTLE_MS, RequiresReady := TRUE) AND Ok;
Ok := M_RegisterConfigDuration(Key := 'press.recipe.transferSettle',
    Item := 'ParCfg/TransferSettleTime', LabelKey := 'project.config.transferSettleTime',
    Kind := E_ConfigKind.PAR_CFG, pTarget := ADR(ParCfg.TransferSettleTime),
    MinimumMs := 0, MaximumMs := RECIPE_MAX_TRANSFER_SETTLE_MS, RequiresReady := TRUE) AND Ok;
Ok := M_RegisterConfigNumber(Key := 'press.recipe.idealCycleMs',
    Item := 'ParCfg/IdealCycleMs', LabelKey := 'project.config.idealCycleMs',
    Unit := E_EngUnit.MILLISECOND, Kind := E_ConfigKind.PAR_CFG,
    Storage := E_ConfigStorage.AS_UDINT, pTarget := ADR(ParCfg.IdealCycleMs),
    Minimum := 0.0, Maximum := 600000.0, RequiresReady := TRUE) AND Ok;
Ok := M_RegisterConfigNumber(Key := 'press.recipe.baselineWorkMs',
    Item := 'ParCfg/BaselineWorkMs', LabelKey := 'project.config.baselineWorkMs',
    Unit := E_EngUnit.MILLISECOND, Kind := E_ConfigKind.PAR_CFG,
    Storage := E_ConfigStorage.AS_UDINT, pTarget := ADR(ParCfg.BaselineWorkMs),
    Minimum := 0.0, Maximum := 600000.0, RequiresReady := TRUE) AND Ok;
Setup := Ok AND PrepareRecipe(Model := InitialModel);
IF Setup THEN CommitRecipe(); END_IF
END_METHOD

// Bind the NC axis for the part-feed servo and arm the module.
//
// Called from OnCyclic until it succeeds, so the axis arms itself the moment an
// NC axis is linked and stays dormant forever on a bench without one. It is
// idempotent and fails closed on both an invalid reference and an unlinked one
// (AxisId 0), which is what makes calling it every scan safe.
//
// The drive is a Jenny Science XENAX Xvi over EtherCAT/CiA402 on the DEV PC's
// own bus - a stand-in for a feed axis, not press cabinet hardware. See the
// note on PartFeedAxis.
//
// The conditions are declared HERE rather than in FB_PressDemoRelease only
// because the axis is not yet in the AUTO chain. When it joins the chain they
// belong beside the other project permits in the Release object, which S7.2.1
// prefers as a single visible component, and this method should shrink to
// binding the reference.
//
// ParCfg limits are deliberately NOT set here. Soft limits, velocity and
// acceleration come from the axis configuration and the recipe (S10.3); a Unit
// that hard-codes a stroke is wrong the first time the mechanics change.
METHOD ConfigurePartFeedAxis : BOOL
VAR_INPUT
    AxisRef : REFERENCE TO AXIS_REF;
END_VAR
IF NOT __ISVALIDREF(AxisRef) THEN
    ConfigurePartFeedAxis := FALSE;
    RETURN;
END_IF
// An AXIS_REF the System Manager has not linked to an NC axis carries AxisId 0.
// This is the test that keeps "absent hardware is absent" true now that arming
// is automatic: without it, a bench with no drive would Setup the module and
// start commanding MC_Power against nothing.
IF AxisRef.NcToPlc.AxisId = 0 THEN
    ConfigurePartFeedAxis := FALSE;
    RETURN;
END_IF
ConfigurePartFeedAxis := PartFeed.Setup(Name := CONCAT(Name, '.PartFeed'),
    AxisRef := AxisRef, Recipe := 0);
IF NOT ConfigurePartFeedAxis THEN
    RETURN;
END_IF
// No project conditions are declared for this axis, and the absence is the
// point rather than an omission. The two that used to be here required the
// press's pneumatic power and its ram guard to be satisfied before the axis
// could move - but the Xvi sits on =000+S-A620, a separate EtherCAT device
// outside the press, with its own power. Neither fact says anything about
// whether that drive may move.
//
// Declaring a condition that does not describe the device is worse than
// declaring none: it blocks motion for a reason the operator cannot act on, and
// it puts a name in the release report that is simply not about this axis
// (S7.2.1 - a condition belongs to the module with the semantic context to own
// it). If this drive is ever mounted INTO a cell, its real conditions get
// declared here then, from that cell's guard and power.
//
// The device-intrinsic gates are untouched and still apply: the axis will not
// jog stale, will not jog while a command owns it, and will not jog without a
// linked NC axis (FB_AxisCM._M_JogCyclic).
// Registered only once it is REAL. A registered child is ticked every scan,
// joins the S8.2 first-out rollup, and appears in the S3.10.2 config walk - and
// therefore in station parameter sets (S3.8b). Registering it unconditionally at
// Setup would put an unnamed module in the published tree and a taught position
// in every saved set for hardware that is not there.
ConfigurePartFeedAxis := _M_Register(PartFeed);
IF NOT ConfigurePartFeedAxis THEN
    RETURN;                            // no free child slot: stay dormant
END_IF
_partFeedConfigured := TRUE;
END_METHOD

END_FUNCTION_BLOCK

// ---- Fraktal_Press_Demo/01_PneumaticPress/Io/FB_PressIoCatalog.TcPOU
// Owner-local I/O engineering-data adapter. This is the ONE source for the approved
// tag/address/description/module-role join. It contains no cyclic behavior,
// process-image access, topology algorithms or device logic.
FUNCTION_BLOCK FB_PressIoCatalog
VAR
    _publisher : FB_IoTopologyPublisher;
    _rootPath : STRING(255);
END_VAR

;

METHOD Setup : BOOL
VAR_INPUT
    UnitRef : REFERENCE TO FB_PressDemoUnit;
    // Core §7.5 register. Only its OUTPUT_FORCING gate can mark a channel
    // Forceable, so a production image publishes Forceable=FALSE everywhere and
    // the HMI renders no force affordance at all (§3.9, §10.5.1 rule 1).
    Engineering : REFERENCE TO FB_EngineeringMode;
END_VAR
VAR
    Ok : BOOL;
    SlideIdentity, DoorIdentity, PressIdentity : ST_CylinderIoIdentity;
    PartIdentity, LowAirIdentity, OperatingAirIdentity : ST_IoPointIdentity;
END_VAR
_rootPath := UnitRef.Name;
Ok := _publisher.Setup(DataRef := GVL_PressFieldbus.Topology, ResetData := TRUE);
Ok := _publisher.M_DefineNode(Index := 1, Name := '=000+S-A610-A1',
    DescriptionKey := 'project.hardware.cx2030', TypeId := 'Beckhoff CX2030',
    Address := 'EtherCAT master', ParentIndex := 0) AND Ok;
Ok := _publisher.M_DefineNode(Index := 2, Name := '=000+S-K010',
    DescriptionKey := 'project.hardware.ek1200', TypeId := 'Beckhoff EK1200-5000',
    Address := 'EtherCAT Box 1', ParentIndex := 1) AND Ok;
Ok := _publisher.M_DefineNode(Index := 3, Name := '=000+S-K010B1',
    DescriptionKey := 'project.hardware.el1809', TypeId := 'Beckhoff EL1809',
    Address := 'EtherCAT Box 2', ParentIndex := 2) AND Ok;
Ok := _publisher.M_DefineNode(Index := 4, Name := '=000+S-K010C1',
    DescriptionKey := 'project.hardware.el2809', TypeId := 'Beckhoff EL2809',
    Address := 'EtherCAT Box 3', ParentIndex := 2) AND Ok;
Ok := _publisher.M_DefineNode(Index := 5, Name := '=000+S-K010D1',
    DescriptionKey := 'project.hardware.el6001', TypeId := 'Beckhoff EL6001 RS232',
    Address := 'EtherCAT Box 4', ParentIndex := 2) AND Ok;
Ok := _publisher.M_DefineNode(Index := 6, Name := '=000+S-K010E',
    DescriptionKey := 'project.hardware.el9011', TypeId := 'Beckhoff EL9011',
    Address := 'EtherCAT Box 5', ParentIndex := 2) AND Ok;

// §10.5.1 — the RS232 terminal's process image. It belongs to no module (nothing
// speaks a protocol over it yet), so its ModulePath is the Unit itself: the bus view
// still shows and forces it, and cross-navigation lands somewhere honest.
Ok := _publisher.M_DefineAnalogChannel(NodeIndex := 5, ChannelIndex := 1,
    Tag := '_000K010D1_Status', DescriptionKey := 'project.io.el6001Status',
    Address := '=000+S-K010D1 Status', Path := '=000+S-K010D1/Status',
    ModulePath := _rootPath, Dir := E_ChannelDir.INPUT, EngUnit := '') AND Ok;
Ok := _publisher.M_DefineAnalogChannel(NodeIndex := 5, ChannelIndex := 2,
    Tag := '_000K010D1_DataIn0', DescriptionKey := 'project.io.el6001DataIn',
    Address := '=000+S-K010D1 Data In 0', Path := '=000+S-K010D1/DataIn0',
    ModulePath := _rootPath, Dir := E_ChannelDir.INPUT, EngUnit := '') AND Ok;
Ok := _publisher.M_DefineAnalogChannel(NodeIndex := 5, ChannelIndex := 3,
    Tag := '_000K010D1_DataIn1', DescriptionKey := 'project.io.el6001DataIn',
    Address := '=000+S-K010D1 Data In 1', Path := '=000+S-K010D1/DataIn1',
    ModulePath := _rootPath, Dir := E_ChannelDir.INPUT, EngUnit := '') AND Ok;
Ok := _publisher.M_DefineAnalogChannel(NodeIndex := 5, ChannelIndex := 4,
    Tag := '_000K010D1_DataIn2', DescriptionKey := 'project.io.el6001DataIn',
    Address := '=000+S-K010D1 Data In 2', Path := '=000+S-K010D1/DataIn2',
    ModulePath := _rootPath, Dir := E_ChannelDir.INPUT, EngUnit := '') AND Ok;
Ok := _publisher.M_DefineAnalogChannel(NodeIndex := 5, ChannelIndex := 5,
    Tag := '_000K010D1_Ctrl', DescriptionKey := 'project.io.el6001Ctrl',
    Address := '=000+S-K010D1 Ctrl', Path := '=000+S-K010D1/Ctrl',
    ModulePath := _rootPath, Dir := E_ChannelDir.OUTPUT, EngUnit := '') AND Ok;
Ok := _publisher.M_DefineAnalogChannel(NodeIndex := 5, ChannelIndex := 6,
    Tag := '_000K010D1_DataOut0', DescriptionKey := 'project.io.el6001DataOut',
    Address := '=000+S-K010D1 Data Out 0', Path := '=000+S-K010D1/DataOut0',
    ModulePath := _rootPath, Dir := E_ChannelDir.OUTPUT, EngUnit := '') AND Ok;
Ok := _publisher.M_DefineAnalogChannel(NodeIndex := 5, ChannelIndex := 7,
    Tag := '_000K010D1_DataOut1', DescriptionKey := 'project.io.el6001DataOut',
    Address := '=000+S-K010D1 Data Out 1', Path := '=000+S-K010D1/DataOut1',
    ModulePath := _rootPath, Dir := E_ChannelDir.OUTPUT, EngUnit := '') AND Ok;
Ok := _publisher.M_DefineAnalogChannel(NodeIndex := 5, ChannelIndex := 8,
    Tag := '_000K010D1_DataOut2', DescriptionKey := 'project.io.el6001DataOut',
    Address := '=000+S-K010D1 Data Out 2', Path := '=000+S-K010D1/DataOut2',
    ModulePath := _rootPath, Dir := E_ChannelDir.OUTPUT, EngUnit := '') AND Ok;

Ok := _M_DefineCylinder(Identity := SlideIdentity,
    ModulePath := UnitRef.PartSlide.Name,
    ExtendedSensorTag := '_101B301A', ExtendedSensorDescription := 'project.io.101B301A',
    ExtendedSensorAddress := '=000+S-K010B1 Ch1', ExtendedSensorIndex := 1,
    RetractedSensorTag := '_101B301B', RetractedSensorDescription := 'project.io.101B301B',
    RetractedSensorAddress := '=000+S-K010B1 Ch2', RetractedSensorIndex := 2,
    ExtendOutputTag := '_101K301A', ExtendOutputDescription := 'project.io.101K301A',
    ExtendOutputAddress := '=000+S-K010C1 Ch1', ExtendOutputIndex := 1,
    RetractOutputTag := '_101K301B', RetractOutputDescription := 'project.io.101K301B',
    RetractOutputAddress := '=000+S-K010C1 Ch2', RetractOutputIndex := 2,
    ExtendedTimeoutKey := 'project.error.slideInsideSensorTimeout',
    RetractedTimeoutKey := 'project.error.slideOutsideSensorTimeout',
    BothSensorsKey := 'project.error.slidePositionSensorsConflict') AND Ok;
UnitRef.PartSlide.ConfigureIoIdentity(Identity := SlideIdentity);
Ok := _M_DefineCylinder(Identity := DoorIdentity,
    ModulePath := UnitRef.Door.Name,
    ExtendedSensorTag := '_101B201A', ExtendedSensorDescription := 'project.io.101B201A',
    ExtendedSensorAddress := '=000+S-K010B1 Ch3', ExtendedSensorIndex := 3,
    RetractedSensorTag := '_101B201B', RetractedSensorDescription := 'project.io.101B201B',
    RetractedSensorAddress := '=000+S-K010B1 Ch4', RetractedSensorIndex := 4,
    ExtendOutputTag := '_101K201A', ExtendOutputDescription := 'project.io.101K201A',
    ExtendOutputAddress := '=000+S-K010C1 Ch3', ExtendOutputIndex := 3,
    RetractOutputTag := '_101K201B', RetractOutputDescription := 'project.io.101K201B',
    RetractOutputAddress := '=000+S-K010C1 Ch4', RetractOutputIndex := 4,
    ExtendedTimeoutKey := 'project.error.doorClosedSensorTimeout',
    RetractedTimeoutKey := 'project.error.doorOpenSensorTimeout',
    BothSensorsKey := 'project.error.doorPositionSensorsConflict') AND Ok;
UnitRef.Door.ConfigureIoIdentity(Identity := DoorIdentity);
Ok := _M_DefineCylinder(Identity := PressIdentity,
    ModulePath := UnitRef.PressRam.Name,
    ExtendedSensorTag := '_101B202A', ExtendedSensorDescription := 'project.io.101B202A',
    ExtendedSensorAddress := '=000+S-K010B1 Ch5', ExtendedSensorIndex := 5,
    RetractedSensorTag := '_101B202B', RetractedSensorDescription := 'project.io.101B202B',
    RetractedSensorAddress := '=000+S-K010B1 Ch6', RetractedSensorIndex := 6,
    ExtendOutputTag := '_101K202A', ExtendOutputDescription := 'project.io.101K202A',
    ExtendOutputAddress := '=000+S-K010C1 Ch5', ExtendOutputIndex := 5,
    RetractOutputTag := '_101K202B', RetractOutputDescription := 'project.io.101K202B',
    RetractOutputAddress := '=000+S-K010C1 Ch6', RetractOutputIndex := 6,
    ExtendedTimeoutKey := 'project.error.pressDownSensorTimeout',
    RetractedTimeoutKey := 'project.error.pressUpSensorTimeout',
    BothSensorsKey := 'project.error.pressPositionSensorsConflict') AND Ok;
UnitRef.PressRam.ConfigureIoIdentity(Identity := PressIdentity);

Ok := _M_DefinePoint(NodeIndex := 3, ChannelIndex := 7, Tag := '_101S101',
    DescriptionKey := 'project.io.101S101', Address := '=000+S-K010B1 Ch7',
    ModulePath := UnitRef.TwoHand.Name, Dir := E_ChannelDir.INPUT) AND Ok;
Ok := _M_DefinePoint(NodeIndex := 3, ChannelIndex := 8, Tag := '_101S102',
    DescriptionKey := 'project.io.101S102', Address := '=000+S-K010B1 Ch8',
    ModulePath := UnitRef.TwoHand.Name, Dir := E_ChannelDir.INPUT) AND Ok;
LowAirIdentity.Tag := '_000MB085A_2';
LowAirIdentity.DescriptionKey := 'project.io.000MB085A_2';
LowAirIdentity.Address := '=000+S-K010B1 Ch10';
LowAirIdentity.ModulePath := UnitRef.AirPressureMonitor.Name;
LowAirIdentity.Path := CONCAT(_rootPath, '.IO._000MB085A_2');
Ok := _M_DefineIdentity(NodeIndex := 3, ChannelIndex := 9,
    Identity := LowAirIdentity, Dir := E_ChannelDir.INPUT) AND Ok;
OperatingAirIdentity.Tag := '_000MB085A_4';
OperatingAirIdentity.DescriptionKey := 'project.io.000MB085A_4';
OperatingAirIdentity.Address := '=000+S-K010B1 Ch11';
OperatingAirIdentity.ModulePath := UnitRef.AirPressureMonitor.Name;
OperatingAirIdentity.Path := CONCAT(_rootPath, '.IO._000MB085A_4');
Ok := _M_DefineIdentity(NodeIndex := 3, ChannelIndex := 10,
    Identity := OperatingAirIdentity, Dir := E_ChannelDir.INPUT) AND Ok;
UnitRef.AirPressureMonitor.ConfigureIoIdentity(LowSensor := LowAirIdentity,
    OperatingSensor := OperatingAirIdentity);
PartIdentity.Tag := '_101B601';
PartIdentity.DescriptionKey := 'project.io.101B601';
PartIdentity.Address := '=000+S-K010B1 Ch12';
PartIdentity.ModulePath := UnitRef.PartPresentSensor.Name;
PartIdentity.Path := CONCAT(_rootPath, '.IO._101B601');
Ok := _M_DefineIdentity(NodeIndex := 3, ChannelIndex := 11,
    Identity := PartIdentity, Dir := E_ChannelDir.INPUT) AND Ok;
UnitRef.PartPresentSensor.ConfigureIoIdentity(Identity := PartIdentity);
Ok := _M_DefinePoint(NodeIndex := 3, ChannelIndex := 12, Tag := '_000K911_Y32',
    DescriptionKey := 'project.io.000K911_Y32', Address := '=000+S-K010B1 Ch14',
    ModulePath := UnitRef.PneumaticPower.Name, Dir := E_ChannelDir.INPUT) AND Ok;
Ok := _M_DefinePoint(NodeIndex := 3, ChannelIndex := 13, Tag := '_000K910A',
    DescriptionKey := 'project.io.000K910A', Address := '=000+S-K010B1 Ch15',
    ModulePath := UnitRef.Name, Dir := E_ChannelDir.INPUT) AND Ok;
Ok := _M_DefinePoint(NodeIndex := 4, ChannelIndex := 7, Tag := '_101P101',
    DescriptionKey := 'project.io.101P101', Address := '=000+S-K010C1 Ch7',
    ModulePath := UnitRef.TwoHand.Name, Dir := E_ChannelDir.OUTPUT) AND Ok;
Ok := _M_DefinePoint(NodeIndex := 4, ChannelIndex := 8, Tag := '_101P102',
    DescriptionKey := 'project.io.101P102', Address := '=000+S-K010C1 Ch8',
    ModulePath := UnitRef.TwoHand.Name, Dir := E_ChannelDir.OUTPUT) AND Ok;
Ok := _M_DefinePoint(NodeIndex := 4, ChannelIndex := 9, Tag := '_000K951_A1',
    DescriptionKey := 'project.io.000K951_A1', Address := '=000+S-K010C1 Ch10',
    ModulePath := UnitRef.PneumaticPower.Name, Dir := E_ChannelDir.OUTPUT) AND Ok;
Ok := _M_DefinePoint(NodeIndex := 4, ChannelIndex := 10, Tag := '_000K911_A1',
    DescriptionKey := 'project.io.000K911_A1', Address := '=000+S-K010C1 Ch11',
    ModulePath := UnitRef.PneumaticPower.Name, Dir := E_ChannelDir.OUTPUT) AND Ok;
Ok := _M_DeclareForceable(Engineering := Engineering) AND Ok;
Setup := _publisher.M_Validate() AND Ok;
END_METHOD

// §3.10.2 - the static fieldbus identity this catalog owns (it set the publisher
// up on it), appended to the owning root's manifest. The Unit reaches the
// topology through the catalog it was given, never through the global itself.
METHOD M_AppendTopologyConfig : BOOL
VAR_INPUT
    Pager : REFERENCE TO FB_ConfigPager;
END_VAR
F_AppendTopologyConfig(Topology := GVL_PressFieldbus.Topology, Pager := Pager);
M_AppendTopologyConfig := TRUE;
END_METHOD

// Core §10.5.1 rule 1 — mark the outputs this station allows to be forced from
// the HMI, and ONLY while the §7.5 OUTPUT_FORCING build gate is active.
//
// Two channels of the EL2809 are deliberately excluded even in a commissioning
// image: =000+S-K010C1 Ch10/Ch11 (_000K951_A1 / _000K911_A1) drive the hardwired
// N54 D2 Control On relay chain. That chain is this machine's control-power
// authority, and §10.5.1 rule 4 keeps the standard-PLC force surface out of
// anything with that role. Forcing them would energize control power from a
// diagnostic screen, which is exactly the act this surface must never offer.
METHOD PRIVATE _M_DeclareForceable : BOOL
VAR_INPUT
    Engineering : REFERENCE TO FB_EngineeringMode;
END_VAR
VAR
    c : INT;
    allow : BOOL;
    Ok : BOOL;
END_VAR
Ok := TRUE;
allow := __ISVALIDREF(Engineering) AND_THEN Engineering.ForcingActive;
// Ch1..Ch8: the six valve coils and the two lamps - actuators whose owning CM
// still runs, still holds its interlocks, and reasserts them the moment the Unit
// leaves the idle MANUAL state that made the force effective (§10.5.1 rule 3).
FOR c := 1 TO 8 DO
    Ok := _publisher.M_SetForceable(NodeIndex := 4, ChannelIndex := c,
        Forceable := allow) AND Ok;
END_FOR
_M_DeclareForceable := Ok;
END_METHOD

// Core §10.5.1 — apply one accepted force request to the approved channel join
// this catalog owns (§10.2.1). Every authority check upstream of the physical
// contract has already happened in FB_UnitBase.ForceChannel; the publisher
// rechecks root ownership, OUTPUT direction and the Forceable capability, and
// refuses anything else. This writes only the held set-point: the hardware
// driver decides each scan whether set-points are applied at all.
METHOD M_RouteForce : BOOL
VAR_INPUT
    ChannelPath : STRING(255);
    OwnerRootPath : STRING(255);
    Force : BOOL;
    BoolValue : BOOL;
    AnalogValue : REAL;
END_VAR
M_RouteForce := _publisher.M_SetForce(ChannelPath := ChannelPath,
    OwnerRootPath := OwnerRootPath, Force := Force,
    BoolValue := BoolValue, AnalogValue := AnalogValue);
END_METHOD

METHOD PRIVATE _M_DefineIdentity : BOOL
VAR_INPUT
    NodeIndex : INT;
    ChannelIndex : INT;
    Identity : ST_IoPointIdentity;
    Dir : E_ChannelDir;
END_VAR
_M_DefineIdentity := _publisher.M_DefineDigitalChannel(
    NodeIndex := NodeIndex, ChannelIndex := ChannelIndex, Tag := Identity.Tag,
    DescriptionKey := Identity.DescriptionKey, Address := Identity.Address,
    Path := Identity.Path, ModulePath := Identity.ModulePath, Dir := Dir);
END_METHOD

METHOD PRIVATE _M_DefinePoint : BOOL
VAR_INPUT
    NodeIndex : INT;
    ChannelIndex : INT;
    Tag : STRING(80);
    DescriptionKey : STRING(160);
    Address : STRING(80);
    ModulePath : STRING(255);
    Dir : E_ChannelDir;
END_VAR
VAR
    Path : STRING(255);
END_VAR
Path := CONCAT(_rootPath, CONCAT('.IO.', Tag));
_M_DefinePoint := _publisher.M_DefineDigitalChannel(NodeIndex := NodeIndex,
    ChannelIndex := ChannelIndex, Tag := Tag, DescriptionKey := DescriptionKey,
    Address := Address, Path := Path, ModulePath := ModulePath, Dir := Dir);
END_METHOD

METHOD PRIVATE _M_DefineCylinder : BOOL
VAR_INPUT
    ModulePath : STRING(255);
    ExtendedSensorTag : STRING(80);
    ExtendedSensorDescription : STRING(160);
    ExtendedSensorAddress : STRING(80);
    ExtendedSensorIndex : INT;
    RetractedSensorTag : STRING(80);
    RetractedSensorDescription : STRING(160);
    RetractedSensorAddress : STRING(80);
    RetractedSensorIndex : INT;
    ExtendOutputTag : STRING(80);
    ExtendOutputDescription : STRING(160);
    ExtendOutputAddress : STRING(80);
    ExtendOutputIndex : INT;
    RetractOutputTag : STRING(80);
    RetractOutputDescription : STRING(160);
    RetractOutputAddress : STRING(80);
    RetractOutputIndex : INT;
    ExtendedTimeoutKey : STRING(255);
    RetractedTimeoutKey : STRING(255);
    BothSensorsKey : STRING(255);
END_VAR
VAR_IN_OUT
    Identity : ST_CylinderIoIdentity;
END_VAR
VAR
    Ok : BOOL;
END_VAR
Identity.ExtendedSensor.Tag := ExtendedSensorTag;
Identity.ExtendedSensor.Address := ExtendedSensorAddress;
Identity.ExtendedSensor.DescriptionKey := ExtendedSensorDescription;
Identity.ExtendedSensor.ModulePath := ModulePath;
Identity.ExtendedSensor.Path := CONCAT(_rootPath, CONCAT('.IO.', ExtendedSensorTag));
Identity.RetractedSensor.Tag := RetractedSensorTag;
Identity.RetractedSensor.Address := RetractedSensorAddress;
Identity.RetractedSensor.DescriptionKey := RetractedSensorDescription;
Identity.RetractedSensor.ModulePath := ModulePath;
Identity.RetractedSensor.Path := CONCAT(_rootPath, CONCAT('.IO.', RetractedSensorTag));
Identity.ExtendOutput.Tag := ExtendOutputTag;
Identity.ExtendOutput.Address := ExtendOutputAddress;
Identity.ExtendOutput.DescriptionKey := ExtendOutputDescription;
Identity.ExtendOutput.ModulePath := ModulePath;
Identity.ExtendOutput.Path := CONCAT(_rootPath, CONCAT('.IO.', ExtendOutputTag));
Identity.RetractOutput.Tag := RetractOutputTag;
Identity.RetractOutput.Address := RetractOutputAddress;
Identity.RetractOutput.DescriptionKey := RetractOutputDescription;
Identity.RetractOutput.ModulePath := ModulePath;
Identity.RetractOutput.Path := CONCAT(_rootPath, CONCAT('.IO.', RetractOutputTag));
Identity.ExtendedTimeoutKey := ExtendedTimeoutKey;
Identity.RetractedTimeoutKey := RetractedTimeoutKey;
Identity.BothSensorsKey := BothSensorsKey;
Ok := _publisher.M_DefineDigitalChannel(NodeIndex := 3, ChannelIndex := ExtendedSensorIndex,
    Tag := Identity.ExtendedSensor.Tag, DescriptionKey := Identity.ExtendedSensor.DescriptionKey,
    Address := Identity.ExtendedSensor.Address, Path := Identity.ExtendedSensor.Path,
    ModulePath := ModulePath, Dir := E_ChannelDir.INPUT);
Ok := _publisher.M_DefineDigitalChannel(NodeIndex := 3, ChannelIndex := RetractedSensorIndex,
    Tag := Identity.RetractedSensor.Tag, DescriptionKey := Identity.RetractedSensor.DescriptionKey,
    Address := Identity.RetractedSensor.Address, Path := Identity.RetractedSensor.Path,
    ModulePath := ModulePath, Dir := E_ChannelDir.INPUT) AND Ok;
Ok := _publisher.M_DefineDigitalChannel(NodeIndex := 4, ChannelIndex := ExtendOutputIndex,
    Tag := Identity.ExtendOutput.Tag, DescriptionKey := Identity.ExtendOutput.DescriptionKey,
    Address := Identity.ExtendOutput.Address, Path := Identity.ExtendOutput.Path,
    ModulePath := ModulePath, Dir := E_ChannelDir.OUTPUT) AND Ok;
Ok := _publisher.M_DefineDigitalChannel(NodeIndex := 4, ChannelIndex := RetractOutputIndex,
    Tag := Identity.RetractOutput.Tag, DescriptionKey := Identity.RetractOutput.DescriptionKey,
    Address := Identity.RetractOutput.Address, Path := Identity.RetractOutput.Path,
    ModulePath := ModulePath, Dir := E_ChannelDir.OUTPUT) AND Ok;
_M_DefineCylinder := Ok;
END_METHOD

END_FUNCTION_BLOCK

// ---- Fraktal_Press_Demo/01_PneumaticPress/Sequences/FB_PressDemoHome.TcPOU
// HOME mode chain (Core §6.2/§6.8 ST skeleton on FB_SequenceBase): establish the
// shared load-safe position, then complete. Finite (does not loop).
FUNCTION_BLOCK FB_PressDemoHome EXTENDS FB_SequenceBase
VAR
    {attribute 'OPC.UA.DA' := '0'}
    _outCmd : REFERENCE TO ST_PneumaticPressOutCmd;
    {attribute 'OPC.UA.DA' := '0'}
    _loadPosition : FB_PressDemoLoadPosition;
END_VAR

METHOD M_Run
IF NOT _attached THEN
    RETURN;
END_IF
CASE _step OF
    0:  // initialize
        M_Step(StepNo := 0, StepName := 'project.step.pressHomeInitialize',
            Awaits := 0, AwaitingLabel := '', TimeClass := E_TimeClass.WORK, ExpectedTime := T#0S, Branch := 0);
        _retVal := E_StepResult.ADVANCE;
        M_Advance(OnAdvance := 900, OnJump1 := -1, OnJump2 := -1, OnJump3 := -1);
    900:  // shared load-safe position (composite step, §6.7)
        _retVal := M_RunSub(Chain := _loadPosition, BaseStepNo := 900);
        M_Advance(OnAdvance := 999, OnJump1 := -1, OnJump2 := -1, OnJump3 := -1);
    999:  // complete
        M_Step(StepNo := 999, StepName := 'project.step.pressHomeComplete',
            Awaits := 0, AwaitingLabel := '', TimeClass := E_TimeClass.WORK, ExpectedTime := T#0S, Branch := 0);
        M_Complete();
ELSE
    M_Fault(Reason := E_Reason.STEP_STALLED, DescriptionKey := 'std.error.undefinedStep');
END_CASE
END_METHOD

METHOD Setup : BOOL
VAR_INPUT
    Host : I_SequenceHost;
END_VAR
VAR_IN_OUT
    PressRam : FB_CylinderCM;
    Door : FB_CylinderCM;
    PartSlide : FB_CylinderCM;
    OutCmd : ST_PneumaticPressOutCmd;
END_VAR
_outCmd REF= OutCmd;
Setup := M_Attach(Host := Host) AND __ISVALIDREF(_outCmd)
    AND _loadPosition.Setup(Host := Host, PressRam := PressRam, Door := Door, PartSlide := PartSlide);
END_METHOD

END_FUNCTION_BLOCK

// ---- Fraktal_Press_Demo/01_PneumaticPress/Sequences/FB_PressDemoLoadPosition.TcPOU
// Shared load-safe-position sub-sequence (Core §6.7): ram up, door open, slide
// outside. HOME and CHANGEOVER both embed it as one composite step, passing a
// BaseStepNo window so its detailed progress projects through the Unit's normal
// §6.5 step record. Implemented as a Core §6.8 ST `CASE _step OF` skeleton on
// FB_SequenceBase — the step actions issue child commands only through the §6.1
// handshake (M_TryIssue), and progression rides the shared _retVal via M_Advance.
FUNCTION_BLOCK FB_PressDemoLoadPosition EXTENDS FB_SequenceBase
VAR
    {attribute 'OPC.UA.DA' := '0'}
    _pressRam : REFERENCE TO FB_CylinderCM;
    {attribute 'OPC.UA.DA' := '0'}
    _door : REFERENCE TO FB_CylinderCM;
    {attribute 'OPC.UA.DA' := '0'}
    _partSlide : REFERENCE TO FB_CylinderCM;
END_VAR

// step body runs via M_Run; the Unit calls this instance each scan

// §6.8 ST step skeleton. One M_Step per step, one commit via M_Advance.
METHOD M_ChainRun
IF NOT _attached THEN
    RETURN;
END_IF
CASE _step OF
    0:  // ram up
        M_Step(StepNo := _baseStepNo, StepName := 'project.step.pressSafePositionRamUp',
            Awaits := _pressRam, AwaitingLabel := 'PressRam.RETRACT',
            TimeClass := E_TimeClass.WORK, ExpectedTime := T#0S, Branch := 0);
        IF M_TryIssue(Steppable := TRUE) THEN
            _pressRam.Abort := FALSE;
            _pressRam.Command := E_CylinderCommand.RETRACT;
            _pressRam.Execute := TRUE;
        END_IF
        IF _pressRam.Done THEN
            _pressRam.Execute := FALSE;
            _retVal := E_StepResult.ADVANCE;
        END_IF
        M_Advance(OnAdvance := 20, OnJump1 := -1, OnJump2 := -1, OnJump3 := -1);
    20:  // door open
        M_Step(StepNo := _baseStepNo + 20, StepName := 'project.step.pressSafePositionDoorOpen',
            Awaits := _door, AwaitingLabel := 'Door.RETRACT',
            TimeClass := E_TimeClass.WORK, ExpectedTime := T#0S, Branch := 0);
        IF M_TryIssue(Steppable := TRUE) THEN
            _door.Abort := FALSE;
            _door.Command := E_CylinderCommand.RETRACT;
            _door.Execute := TRUE;
        END_IF
        IF _door.Done THEN
            _door.Execute := FALSE;
            _retVal := E_StepResult.ADVANCE;
        END_IF
        M_Advance(OnAdvance := 40, OnJump1 := -1, OnJump2 := -1, OnJump3 := -1);
    40:  // slide outside
        M_Step(StepNo := _baseStepNo + 40, StepName := 'project.step.pressSafePositionSlideOutside',
            Awaits := _partSlide, AwaitingLabel := 'PartSlide.RETRACT',
            TimeClass := E_TimeClass.WORK, ExpectedTime := T#0S, Branch := 0);
        IF M_TryIssue(Steppable := TRUE) THEN
            _partSlide.Abort := FALSE;
            _partSlide.Command := E_CylinderCommand.RETRACT;
            _partSlide.Execute := TRUE;
        END_IF
        IF _partSlide.Done THEN
            _partSlide.Execute := FALSE;
            _retVal := E_StepResult.ADVANCE;
        END_IF
        M_Advance(OnAdvance := 999, OnJump1 := -1, OnJump2 := -1, OnJump3 := -1);
    999:  // established
        M_Step(StepNo := _baseStepNo + 60, StepName := 'project.step.pressSafePositionComplete',
            Awaits := 0, AwaitingLabel := '', TimeClass := E_TimeClass.WORK, ExpectedTime := T#0S, Branch := 0);
        Done := TRUE;
ELSE
    M_Fault(Reason := E_Reason.STEP_STALLED, DescriptionKey := 'std.error.undefinedStep');
END_CASE
END_METHOD

METHOD Setup : BOOL
VAR_INPUT
    Host : I_SequenceHost;
END_VAR
VAR_IN_OUT
    PressRam : FB_CylinderCM;
    Door : FB_CylinderCM;
    PartSlide : FB_CylinderCM;
END_VAR
_pressRam REF= PressRam;
_door REF= Door;
_partSlide REF= PartSlide;
Setup := M_Attach(Host := Host)
    AND __ISVALIDREF(_pressRam) AND __ISVALIDREF(_door) AND __ISVALIDREF(_partSlide);
END_METHOD

END_FUNCTION_BLOCK

// ---- Fraktal_Press_Demo/01_PneumaticPress/Sequences/FB_PressDemoChangeover.TcPOU
// CHANGEOVER mode chain (Core §6.2/§6.8 ST skeleton on FB_SequenceBase): validate
// the selected model, establish the shared load-safe position, then ask the
// operator (§6.11) to confirm tooling/material match before completing. The
// 'repeat position' answer restarts the guided move via a backward jump (§6.10).
FUNCTION_BLOCK FB_PressDemoChangeover EXTENDS FB_SequenceBase
VAR
    _decisionRequest : ST_DecisionRequest;
    _answer : INT;
    _modelSelected : BOOL;
    {attribute 'OPC.UA.DA' := '0'}
    _outCmd : REFERENCE TO ST_PneumaticPressOutCmd;
    {attribute 'OPC.UA.DA' := '0'}
    _model : REFERENCE TO ST_ModelId;
    {attribute 'OPC.UA.DA' := '0'}
    _loadPosition : FB_PressDemoLoadPosition;
END_VAR

// §6.8 - the chain's own state on a restart (the base resets the flow state).
METHOD PROTECTED OnChainReset
_answer := 0;
END_METHOD

METHOD M_Run
IF NOT _attached THEN
    RETURN;
END_IF
CASE _step OF
    0:  // initialize
        M_Step(StepNo := 0, StepName := 'project.step.pressChangeoverInitialize',
            Awaits := 0, AwaitingLabel := '', TimeClass := E_TimeClass.WORK, ExpectedTime := T#0S, Branch := 0);
        _outCmd.ChangeoverCompleted := FALSE;
        _answer := 0;
        _decisionRequest.Prompt := '';
        M_ClearDecision();
        _retVal := E_StepResult.ADVANCE;
        M_Advance(OnAdvance := 800, OnJump1 := -1, OnJump2 := -1, OnJump3 := -1);
    800:  // validate the transactionally-loaded model
        M_Step(StepNo := 800, StepName := 'project.step.pressChangeoverValidateModel',
            Awaits := 0, AwaitingLabel := '', TimeClass := E_TimeClass.WAIT_OPERATOR, ExpectedTime := T#0S, Branch := 0);
        _modelSelected := M_Await(Idx := 1, Label := 'project.condition.pressModelSelected',
            Ok := _model.ModelCode <> '');
        IF _modelSelected THEN
            _retVal := E_StepResult.ADVANCE;
        END_IF
        M_Advance(OnAdvance := 810, OnJump1 := -1, OnJump2 := -1, OnJump3 := -1);
    810:  // shared load-safe position (composite step)
        _retVal := M_RunSub(Chain := _loadPosition, BaseStepNo := 810);
        M_Advance(OnAdvance := 870, OnJump1 := -1, OnJump2 := -1, OnJump3 := -1);
    870:  // request tooling/material confirmation
        M_Step(StepNo := 870, StepName := 'project.step.pressChangeoverRequestConfirmation',
            Awaits := 0, AwaitingLabel := '', TimeClass := E_TimeClass.WAIT_OPERATOR, ExpectedTime := T#0S, Branch := 0);
        _decisionRequest.Prompt := 'project.decision.pressChangeoverConfirm';
        _decisionRequest.Options[1] := 'project.decision.confirmChangeover';
        _decisionRequest.Options[2] := 'project.decision.repeatChangeoverPosition';
        _decisionRequest.Default := 0;
        _decisionRequest.Timeout := T#0S;
        M_AskDecision(Req := _decisionRequest);
        _retVal := E_StepResult.ADVANCE;
        M_Advance(OnAdvance := 880, OnJump1 := -1, OnJump2 := -1, OnJump3 := -1);
    880:  // await confirmation; JUMP1 = repeat the guided position
        M_Step(StepNo := 880, StepName := 'project.step.pressChangeoverAwaitConfirmation',
            Awaits := 0, AwaitingLabel := '', TimeClass := E_TimeClass.WAIT_OPERATOR, ExpectedTime := T#0S, Branch := 0);
        _answer := M_TakeDecision();
        IF _answer = 1 THEN
            _retVal := E_StepResult.ADVANCE;
        ELSIF _answer = 2 THEN
            _retVal := E_StepResult.JUMP1;
        ELSE
            _modelSelected := M_Await(Idx := 1,
                Label := 'project.condition.pressChangeoverConfirmation', Ok := FALSE);
        END_IF
        M_Advance(OnAdvance := 999, OnJump1 := 810, OnJump2 := -1, OnJump3 := -1);
    999:  // complete
        M_Step(StepNo := 999, StepName := 'project.step.pressChangeoverComplete',
            Awaits := 0, AwaitingLabel := '', TimeClass := E_TimeClass.WORK, ExpectedTime := T#0S, Branch := 0);
        _outCmd.ChangeoverCompleted := TRUE;
        M_Complete();
ELSE
    M_Fault(Reason := E_Reason.STEP_STALLED, DescriptionKey := 'std.error.undefinedStep');
END_CASE
END_METHOD

METHOD Setup : BOOL
VAR_INPUT
    Host : I_SequenceHost;
END_VAR
VAR_IN_OUT
    PressRam : FB_CylinderCM;
    Door : FB_CylinderCM;
    PartSlide : FB_CylinderCM;
    OutCmd : ST_PneumaticPressOutCmd;
    Model : ST_ModelId;
END_VAR
_outCmd REF= OutCmd;
_model REF= Model;
Setup := M_Attach(Host := Host) AND __ISVALIDREF(_outCmd) AND __ISVALIDREF(_model)
    AND _loadPosition.Setup(Host := Host, PressRam := PressRam, Door := Door, PartSlide := PartSlide);
END_METHOD

END_FUNCTION_BLOCK

// ---- Fraktal_Press_Demo/01_PneumaticPress/Sequences/FB_PressDemoAuto.TcPOU
// AUTO mode chain (Core §6.2/§6.8 ST skeleton on FB_SequenceBase): the continuous
// production cycle — await a fresh two-hand start with part+air present, transfer
// the part in, press for the recipe dwell, return to load position, count the good
// part, and loop until Stop. A Stop requested at the between-cycles wait is honored
// there (M_StopNow) so no phantom cycle is charged. Every child motion goes through
// the §6.1 handshake (M_TryIssue); progression rides the shared _retVal.
FUNCTION_BLOCK FB_PressDemoAuto EXTENDS FB_SequenceBase
VAR
    _partReady, _airReady, _startReady : BOOL;
    _dwellTwoHandHeld : BOOL;          // N220 named wait: two-hand held through the dwell
    _decisionRequest : ST_DecisionRequest;   // §6.11 not-reached confirmation
    _answer : INT;
    _ramReached, _failureConfirmed : BOOL;   // N200/N210 named waits
    _twoHandHeldDuringClose : BOOL;          // N180 named wait
    _closeAbortWarned : BOOL;                // N180 §6.9(e) message result
    _ramFailureReported : BOOL;              // N200 §6.9(e) message result
    _partInMachine : BOOL;                   // §3.16.3 the part is already received
    _partDispositioned : BOOL;               // N260 already set the verdict
    _traceAccepted, _recordAccepted, _partProcessed : BOOL;
    {attribute 'OPC.UA.DA' := '0'}
    _pressRam : REFERENCE TO FB_CylinderCM;
    {attribute 'OPC.UA.DA' := '0'}
    _door : REFERENCE TO FB_CylinderCM;
    {attribute 'OPC.UA.DA' := '0'}
    _partSlide : REFERENCE TO FB_CylinderCM;
    {attribute 'OPC.UA.DA' := '0'}
    _twoHand : REFERENCE TO FB_TwoHandStartCM;
    {attribute 'OPC.UA.DA' := '0'}
    _partPresentSensor : REFERENCE TO FB_DigitalInputCM;
    {attribute 'OPC.UA.DA' := '0'}
    _airPressureMonitor : REFERENCE TO FB_AirPressureMonitorCM;
    {attribute 'OPC.UA.DA' := '0'}
    _parCfg : REFERENCE TO ST_PneumaticPressParCfg;
    // §3.8a - the CELL's own policy, held separately from the MODEL's data and
    // referenced exactly like _parCfg, so each step reads whichever structure
    // actually owns the value it is asking about.
    {attribute 'OPC.UA.DA' := '0'}
    _stationCfg : REFERENCE TO ST_PneumaticPressStationCfg;
    {attribute 'OPC.UA.DA' := '0'}
    _outCmd : REFERENCE TO ST_PneumaticPressOutCmd;
    {attribute 'OPC.UA.DA' := '0'}
    _startLatched : REFERENCE TO BOOL;
    {attribute 'OPC.UA.DA' := '0'}
    _loadPosition : FB_PressDemoLoadPosition;
END_VAR

// §6.8 - the chain's own state on a restart (the base resets the flow state).
METHOD PROTECTED OnChainReset
// A chart restart abandons whatever the cycle was holding: the part record is
// closed by N215/N999, never by a restart, so both trackers start clean.
_partDispositioned := FALSE;
_partInMachine := FALSE;
END_METHOD

